(* IEC 61131-3 sources: RL_MAR/experiments/results/ablation/Ablation_no_post_process_deepseek-ai_DeepSeek-V3.2_20260602_235132, 94 files *)

(* ---- hard_92.st ---- *)
TYPE
    ST_BreakerStatus :
    STRUCT
        Opened : BOOL;
        Closed : BOOL;
    END_STRUCT;

    ST_BreakerControl :
    STRUCT
        Trip : BOOL;
        Close : BOOL;
    END_STRUCT;

    ST_BreakerData :
    STRUCT
        Control : ST_BreakerControl;
        Status : ST_BreakerStatus;
    END_STRUCT;

    ST_PointData :
    STRUCT
        Point_1a : INT;
        Point_2a : INT;
        Point_3a : INT;
        Point_4a : INT;
    END_STRUCT;

    E_BreakerID :
    (
        B10_1,
        B10_2,
        B10_12,
        B54,
        B55,
        B56,
        B57
    );
END_TYPE

FUNCTION_BLOCK FB_BreakerControlSystem
VAR_INPUT
    B10_1_Trip : BOOL;
    B10_1_Close : BOOL;
    B10_2_Trip : BOOL;
    B10_2_Close : BOOL;
    B10_12_Trip : BOOL;
    B10_12_Close : BOOL;
    B54_Trip : BOOL;
    B54_Close : BOOL;
    B55_Trip : BOOL;
    B55_Close : BOOL;
    B56_Trip : BOOL;
    B56_Close : BOOL;
    B57_Trip : BOOL;
    B57_Close : BOOL;
END_VAR

VAR_OUTPUT
    Point_1a : INT;
    Point_2a : INT;
    Point_3a : INT;
    Point_4a : INT;
    B10_1_Opened : BOOL;
    B10_1_Closed : BOOL;
    B10_2_Opened : BOOL;
    B10_2_Closed : BOOL;
    B10_12_Opened : BOOL;
    B10_12_Closed : BOOL;
    B54_Opened : BOOL;
    B54_Closed : BOOL;
    B55_Opened : BOOL;
    B55_Closed : BOOL;
    B56_Opened : BOOL;
    B56_Closed : BOOL;
    B57_Opened : BOOL;
    B57_Closed : BOOL;
END_VAR

VAR
    // Internal structured data storage for breakers and points
    rBreakers : ARRAY[E_BreakerID] OF ST_BreakerData;
    rPoints : ST_PointData;
    // Intermediate condition variables
    bCondition_1A : BOOL;
    bCondition_2A : BOOL;
    // Internal variables as per original specification (initialized but not used in core logic)
    SEL86_OUT : INT;
    MOVE89_OUT : INT;
    SEL66_OUT : INT;
    MOVE69_OUT : INT;
    SEL96_OUT : INT;
    MOVE99_OUT : INT;
    SEL106_OUT : INT;
    MOVE109_OUT : INT;
END_VAR

// Main Execution Logic
// Step 1: Update all breaker states based on control signals
// Breaker B10_1
IF rBreakers[B10_1].Control.Close <> B10_1_Close THEN
    rBreakers[B10_1].Control.Close := B10_1_Close;
END_IF;
IF rBreakers[B10_1].Control.Trip <> B10_1_Trip THEN
    rBreakers[B10_1].Control.Trip := B10_1_Trip;
END_IF;

IF B10_1_Close THEN
    rBreakers[B10_1].Status.Closed := TRUE;
    rBreakers[B10_1].Status.Opened := FALSE;
ELSIF B10_1_Trip THEN
    rBreakers[B10_1].Status.Closed := FALSE;
    rBreakers[B10_1].Status.Opened := TRUE;
END_IF;

// Breaker B10_2
IF rBreakers[B10_2].Control.Close <> B10_2_Close THEN
    rBreakers[B10_2].Control.Close := B10_2_Close;
END_IF;
IF rBreakers[B10_2].Control.Trip <> B10_2_Trip THEN
    rBreakers[B10_2].Control.Trip := B10_2_Trip;
END_IF;

IF B10_2_Close THEN
    rBreakers[B10_2].Status.Closed := TRUE;
    rBreakers[B10_2].Status.Opened := FALSE;
ELSIF B10_2_Trip THEN
    rBreakers[B10_2].Status.Closed := FALSE;
    rBreakers[B10_2].Status.Opened := TRUE;
END_IF;

// Breaker B10_12
IF rBreakers[B10_12].Control.Close <> B10_12_Close THEN
    rBreakers[B10_12].Control.Close := B10_12_Close;
END_IF;
IF rBreakers[B10_12].Control.Trip <> B10_12_Trip THEN
    rBreakers[B10_12].Control.Trip := B10_12_Trip;
END_IF;

IF B10_12_Close THEN
    rBreakers[B10_12].Status.Closed := TRUE;
    rBreakers[B10_12].Status.Opened := FALSE;
ELSIF B10_12_Trip THEN
    rBreakers[B10_12].Status.Closed := FALSE;
    rBreakers[B10_12].Status.Opened := TRUE;
END_IF;

// Breaker B54
IF rBreakers[B54].Control.Close <> B54_Close THEN
    rBreakers[B54].Control.Close := B54_Close;
END_IF;
IF rBreakers[B54].Control.Trip <> B54_Trip THEN
    rBreakers[B54].Control.Trip := B54_Trip;
END_IF;

IF B54_Close THEN
    rBreakers[B54].Status.Closed := TRUE;
    rBreakers[B54].Status.Opened := FALSE;
ELSIF B54_Trip THEN
    rBreakers[B54].Status.Closed := FALSE;
    rBreakers[B54].Status.Opened := TRUE;
END_IF;

// Breaker B55
IF rBreakers[B55].Control.Close <> B55_Close THEN
    rBreakers[B55].Control.Close := B55_Close;
END_IF;
IF rBreakers[B55].Control.Trip <> B55_Trip THEN
    rBreakers[B55].Control.Trip := B55_Trip;
END_IF;

IF B55_Close THEN
    rBreakers[B55].Status.Closed := TRUE;
    rBreakers[B55].Status.Opened := FALSE;
ELSIF B55_Trip THEN
    rBreakers[B55].Status.Closed := FALSE;
    rBreakers[B55].Status.Opened := TRUE;
END_IF;

// Breaker B56
IF rBreakers[B56].Control.Close <> B56_Close THEN
    rBreakers[B56].Control.Close := B56_Close;
END_IF;
IF rBreakers[B56].Control.Trip <> B56_Trip THEN
    rBreakers[B56].Control.Trip := B56_Trip;
END_IF;

IF B56_Close THEN
    rBreakers[B56].Status.Closed := TRUE;
    rBreakers[B56].Status.Opened := FALSE;
ELSIF B56_Trip THEN
    rBreakers[B56].Status.Closed := FALSE;
    rBreakers[B56].Status.Opened := TRUE;
END_IF;

// Breaker B57
IF rBreakers[B57].Control.Close <> B57_Close THEN
    rBreakers[B57].Control.Close := B57_Close;
END_IF;
IF rBreakers[B57].Control.Trip <> B57_Trip THEN
    rBreakers[B57].Control.Trip := B57_Trip;
END_IF;

IF B57_Close THEN
    rBreakers[B57].Status.Closed := TRUE;
    rBreakers[B57].Status.Opened := FALSE;
ELSIF B57_Trip THEN
    rBreakers[B57].Status.Closed := FALSE;
    rBreakers[B57].Status.Opened := TRUE;
END_IF;

// Step 2: Calculate intermediate conditions
bCondition_1A := (rBreakers[B10_12].Status.Closed AND rBreakers[B10_1].Status.Closed) OR rBreakers[B10_2].Status.Closed;
bCondition_2A := (rBreakers[B10_12].Status.Closed AND rBreakers[B10_2].Status.Closed) OR rBreakers[B10_1].Status.Closed;

// Step 3: Calculate output points
// Point_1a
IF rBreakers[B54].Status.Closed AND bCondition_1A THEN
    rPoints.Point_1a := 0;
ELSE
    rPoints.Point_1a := 138;
END_IF;

// Point_2a
IF rBreakers[B55].Status.Closed AND bCondition_1A THEN
    rPoints.Point_2a := 0;
ELSE
    rPoints.Point_2a := 138;
END_IF;

// Point_3a
IF rBreakers[B56].Status.Closed AND bCondition_2A THEN
    rPoints.Point_3a := 0;
ELSE
    rPoints.Point_3a := 138;
END_IF;

// Point_4a
IF rBreakers[B57].Status.Closed AND bCondition_2A THEN
    rPoints.Point_4a := 0;
ELSE
    rPoints.Point_4a := 138;
END_IF;

// Step 4: Map internal data to public outputs
Point_1a := rPoints.Point_1a;
Point_2a := rPoints.Point_2a;
Point_3a := rPoints.Point_3a;
Point_4a := rPoints.Point_4a;

B10_1_Opened := rBreakers[B10_1].Status.Opened;
B10_1_Closed := rBreakers[B10_1].Status.Closed;
B10_2_Opened := rBreakers[B10_2].Status.Opened;
B10_2_Closed := rBreakers[B10_2].Status.Closed;
B10_12_Opened := rBreakers[B10_12].Status.Opened;
B10_12_Closed := rBreakers[B10_12].Status.Closed;
B54_Opened := rBreakers[B54].Status.Opened;
B54_Closed := rBreakers[B54].Status.Closed;
B55_Opened := rBreakers[B55].Status.Opened;
B55_Closed := rBreakers[B55].Status.Closed;
B56_Opened := rBreakers[B56].Status.Opened;
B56_Closed := rBreakers[B56].Status.Closed;
B57_Opened := rBreakers[B57].Status.Opened;
B57_Closed := rBreakers[B57].Status.Closed;

// Step 5: Initialize internal placeholder variables (as per original spec)
SEL86_OUT := 0;
MOVE89_OUT := 0;
SEL66_OUT := 0;
MOVE69_OUT := 0;
SEL96_OUT := 0;
MOVE99_OUT := 0;
SEL106_OUT := 0;
MOVE109_OUT := 0;

END_FUNCTION_BLOCK

(* ---- hard_93.st ---- *)
FUNCTION_BLOCK FB_CircuitControl
VAR_INPUT
    Reset_All_CB : BOOL;
    Current_Fault_on_TRSF1 : INT;
    Current_Fault_on_66BUS1 : INT;
END_VAR

VAR_OUTPUT
    Short_Circuit_TRSF1 : BOOL;
    Short_Circuit_66BUS : BOOL;
    Open_CB1_66KV : BOOL;
    Open_CB2_66KV : BOOL;
    Open_CB_TRSF1 : BOOL;
    Open_CB2_22KV : BOOL;
END_VAR

VAR
    Threshold500 : INT := 500;
    Prev_Open_CB2_22KV : BOOL;
    Prev_Open_CB1_66KV : BOOL;
    Prev_Open_CB_TRSF1 : BOOL;
    bTemp_Open_CB2_22KV : BOOL;
    bTemp_Open_CB1_66KV : BOOL;
    bTemp_Open_CB_TRSF1 : BOOL;
END_VAR

(* Part a: Short circuit detection *)
Short_Circuit_66BUS := (Current_Fault_on_66BUS1 > Threshold500);
Short_Circuit_TRSF1 := (Current_Fault_on_TRSF1 > Threshold500);

(* Part b: Circuit breaker control logic *)
(* Reset condition takes highest priority *)
IF Reset_All_CB THEN
    Open_CB1_66KV := FALSE;
    Open_CB2_66KV := FALSE;
    Open_CB_TRSF1 := FALSE;
    Open_CB2_22KV := FALSE;
    Prev_Open_CB2_22KV := FALSE;
    Prev_Open_CB1_66KV := FALSE;
    Prev_Open_CB_TRSF1 := FALSE;
ELSE
    (* Open_CB2_66KV is always TRUE (closed) per specification *)
    Open_CB2_66KV := TRUE;

    (* First pass: Initial calculations using previous cycle states *)
    bTemp_Open_CB2_22KV := (NOT Prev_Open_CB2_22KV) AND
                           ((Open_CB1_66KV AND Open_CB_TRSF1) OR Short_Circuit_66BUS);

    bTemp_Open_CB1_66KV := (NOT bTemp_Open_CB2_22KV) AND
                           ((Prev_Open_CB1_66KV AND Open_CB_TRSF1) OR Short_Circuit_66BUS);

    bTemp_Open_CB_TRSF1 := (NOT bTemp_Open_CB2_22KV) AND
                           ((Open_CB1_66KV AND Prev_Open_CB_TRSF1) OR Short_Circuit_66BUS);

    (* Second pass: Update calculations using intermediate values *)
    bTemp_Open_CB2_22KV := bTemp_Open_CB2_22KV OR
                          ((NOT Prev_Open_CB2_22KV) AND
                           ((Open_CB2_66KV AND bTemp_Open_CB1_66KV AND bTemp_Open_CB_TRSF1) OR Short_Circuit_TRSF1));

    bTemp_Open_CB1_66KV := bTemp_Open_CB1_66KV OR
                          ((NOT bTemp_Open_CB2_22KV) AND
                           ((Open_CB2_66KV AND Prev_Open_CB1_66KV AND bTemp_Open_CB_TRSF1) OR Short_Circuit_TRSF1));

    bTemp_Open_CB_TRSF1 := bTemp_Open_CB_TRSF1 OR
                          ((NOT bTemp_Open_CB2_22KV) AND
                           ((Open_CB2_66KV AND bTemp_Open_CB1_66KV AND Prev_Open_CB_TRSF1) OR Short_Circuit_TRSF1));

    (* Assign final values to outputs *)
    Open_CB2_22KV := bTemp_Open_CB2_22KV;
    Open_CB1_66KV := bTemp_Open_CB1_66KV;
    Open_CB_TRSF1 := bTemp_Open_CB_TRSF1;

    (* Store current states for next scan cycle *)
    Prev_Open_CB2_22KV := Open_CB2_22KV;
    Prev_Open_CB1_66KV := Open_CB1_66KV;
    Prev_Open_CB_TRSF1 := Open_CB_TRSF1;
END_IF;

END_FUNCTION_BLOCK;

(* ---- hard_94.st ---- *)
FUNCTION_BLOCK FB_AdvancedCircuitBreakerControl
VAR_INPUT
    S_AL1_P_B1 : BOOL;
    S_AL1_P_B2 : BOOL;
    S_AL1_MCB : BOOL;
    MCB_BUSY : BOOL;
    MCB_ERROR : BOOL;
    S_AL1_MCBR : BOOL;
    MCBR_BUSY : BOOL;
    MCBR_ERROR : BOOL;
    S_AL1_P_B3 : BOOL;
    S_AL1_MCB2 : BOOL;
    S_AL1_MCBR2 : BOOL;
END_VAR
VAR_OUTPUT
    E_AL1_B1 : BOOL;
    PUWS_AL1_B1_PLUS : BOOL;
    PUWS_AL1_B1_RIGHT : BOOL;
    PAS_AL1_PLUS : BOOL;
    PAS_AL1_TURN : BOOL;
END_VAR
VAR
    (* State Variables - Only one should be active at a time *)
    PPAL1 : BOOL := 1;
    PP0 : BOOL := 0;
    PP1 : BOOL := 0;
    PP2 : BOOL := 0;
    PP3 : BOOL := 0;
    PP4 : BOOL := 0;
    PP5 : BOOL := 0;
    PP7 : BOOL := 0;
    PPL3 : BOOL := 0;
    PPL4 : BOOL := 0;
    PPL5 : BOOL := 0;
    PPL7 : BOOL := 0;

    (* Internal Control and Status Flags *)
    MCB : BOOL := 1;
    MCBR : BOOL := 1;
    MCB_CONTROL : BOOL;
    STABLE : BOOL;
END_VAR

(* Main State Machine Logic *)
STABLE := 0;
WHILE (STABLE = 0) DO
    STABLE := 1;

    (* State PP0 to PP1 *)
    IF (PP0 = 1) AND (NOT MCB_CONTROL) AND (PP1 = 0) THEN
        PP0 := 0;
        PP1 := 1;
        STABLE := 0;
    END_IF;

    (* State PP1 to PP2 *)
    IF (PP1 = 1) AND S_AL1_P_B1 AND (PP2 = 0) THEN
        PP1 := 0;
        PP2 := 1;
        STABLE := 0;
    END_IF;

    (* State PP2 to PP3 (Main Path) *)
    IF (PP2 = 1) AND S_AL1_P_B2 AND (NOT MCB_CONTROL) AND (PP3 = 0) THEN
        PP2 := 0;
        PP3 := 1;
        STABLE := 0;
    END_IF;

    (* State PP2 to PPL3 (Alternative Path) *)
    IF (PP2 = 1) AND S_AL1_P_B2 AND MCB_CONTROL AND (PPL3 = 0) AND (PP1 = 0) THEN
        PP2 := 0;
        PPL3 := 1;
        PP1 := 1;
        STABLE := 0;
    END_IF;

    (* State PP3 to PP4 *)
    IF (PP3 = 1) AND S_AL1_MCB AND (PP4 = 0) AND (PP1 = 0) THEN
        PP3 := 0;
        PP4 := 1;
        PP1 := 1;
        STABLE := 0;
    END_IF;

    (* State PP4 to PP5 *)
    IF (PP4 = 1) AND (MCB = 1) AND MCB_BUSY AND (PP5 = 0) THEN
        PP4 := 0;
        MCB := 0;
        PP5 := 1;
        STABLE := 0;
    END_IF;

    (* State PP5 to PP7 *)
    IF (PP5 = 1) AND S_AL1_MCB2 AND (PP7 = 0) AND (MCB = 0) THEN
        PP5 := 0;
        PP7 := 1;
        MCB := 1;
        STABLE := 0;
    END_IF;

    (* State PP7 to End *)
    IF (PP7 = 1) AND S_AL1_P_B3 THEN
        PP7 := 0;
        STABLE := 0;
    END_IF;

    (* State PPL3 to PPL4 *)
    IF (PPL3 = 1) AND S_AL1_MCBR AND (PPL4 = 0) THEN
        PPL3 := 0;
        PPL4 := 1;
        STABLE := 0;
    END_IF;

    (* State PPL4 to PPL5 *)
    IF (PPL4 = 1) AND (MCBR = 1) AND MCBR_BUSY AND (PPL5 = 0) THEN
        PPL4 := 0;
        MCBR := 0;
        PPL5 := 1;
        STABLE := 0;
    END_IF;

    (* State PPL5 to PPL7 *)
    IF (PPL5 = 1) AND S_AL1_MCBR2 AND (PPL7 = 0) AND (MCBR = 0) THEN
        PPL5 := 0;
        PPL7 := 1;
        MCBR := 1;
        STABLE := 0;
    END_IF;

    (* State PPL7 to End *)
    IF (PPL7 = 1) AND S_AL1_P_B3 THEN
        PPL7 := 0;
        STABLE := 0;
    END_IF;
END_WHILE;

(* Output Control Logic *)
(* Initialize all outputs to FALSE *)
E_AL1_B1 := 0;
PUWS_AL1_B1_PLUS := 0;
PUWS_AL1_B1_RIGHT := 0;
PAS_AL1_PLUS := 0;
PAS_AL1_TURN := 0;
MCB_CONTROL := 0;

(* Set outputs based on active states *)
IF (PP0 = 1) OR (PP1 = 1) THEN
    E_AL1_B1 := 1;
END_IF;

IF (PP3 = 1) THEN
    MCB_CONTROL := 1;
END_IF;

IF (PPL3 = 1) OR (PPL4 = 1) THEN
    PAS_AL1_PLUS := 1;
    PAS_AL1_TURN := 1;
END_IF;

IF (PPAL1 = 1) OR (PP2 = 1) THEN
    PUWS_AL1_B1_PLUS := 1;
END_IF;

IF (PP2 = 1) OR (PP3 = 1) OR (PPL3 = 1) THEN
    E_AL1_B1 := 0;
END_IF;

IF (PP0 = 1) OR (PP3 = 1) THEN
    MCB_CONTROL := 0;
END_IF;

IF (PP0 = 1) OR (PP3 = 1) OR (PP4 = 1) THEN
    PAS_AL1_PLUS := 0;
    PAS_AL1_TURN := 0;
END_IF;

IF (PPAL1 = 1) OR (PP2 = 1) THEN
    PUWS_AL1_B1_RIGHT := 0;
END_IF;

END_FUNCTION_BLOCK

(* ---- hf_1.st ---- *)
FUNCTION_BLOCK StackMin
VAR_INPUT
    push : BOOL;
    pop : BOOL;
    reset : BOOL;
END_VAR
VAR_OUTPUT
    error : BOOL;
    status : WORD;
END_VAR
VAR_IN_OUT
    item : INT;
    stack : ARRAY[0..3] OF INT;
END_VAR
VAR
    top : INT := -1;
    i : INT;
    minIndex : INT;
    minValue : INT;
END_VAR

(* Reset has highest priority *)
IF reset THEN
    top := -1;
    error := FALSE;
    status := 16#0000;
ELSIF push THEN
    (* Push operation *)
    IF top >= 3 THEN
        error := TRUE;
        status := 16#8A04;
    ELSE
        top := top + 1;
        stack[top] := item;
        error := FALSE;
        status := 16#0000;
    END_IF;
ELSIF pop THEN
    (* Pop-minimum operation *)
    IF top < 0 THEN
        error := TRUE;
        status := 16#8A05;
    ELSE
        (* Find minimum value and its index *)
        minIndex := 0;
        minValue := stack[0];
        FOR i := 1 TO top DO
            IF stack[i] < minValue THEN
                minValue := stack[i];
                minIndex := i;
            END_IF;
        END_FOR;

        (* Output the minimum value *)
        item := minValue;

        (* Shift elements down to remove the minimum *)
        FOR i := minIndex TO top - 1 DO
            stack[i] := stack[i + 1];
        END_FOR;

        (* Decrement top index *)
        top := top - 1;

        error := FALSE;
        status := 16#0000;
    END_IF;
ELSE
    (* No operation - maintain current state *)
    error := FALSE;
    status := 16#0000;
END_IF;

END_FUNCTION_BLOCK

(* ---- hf_10.st ---- *)
TYPE
    // Define a circular buffer structure for clarity and maintainability
    CircularBuffer : STRUCT
        Data : ARRAY[1..100] OF REAL;
        Head : INT; // Points to the oldest element (next to be overwritten)
        Count : INT; // Number of valid elements currently in the buffer
        Sum : REAL;
    END_STRUCT;
END_TYPE

FUNCTION_BLOCK FloatingAverage
VAR_INPUT
    cyclicExecution : BOOL; // When TRUE, periodic reading is performed, and trigger has no effect
    trigger : BOOL; // External trigger signal, reads value upon each rising edge
    value : REAL; // Newly read data value
    windowSize : INT; // The window size for the moving average, which must be between 1 and 100
    reset : BOOL; // Reset signal, resets the moving average calculation when TRUE
END_VAR
VAR_OUTPUT
    average : REAL; // The moving average
    windowSizeReached : BOOL; // FALSE: Maximum window width not yet reached, TRUE: Maximum window width has been reached
    error : BOOL; // FALSE: No error occurred, TRUE: An error occurred during the execution of FB
    status : WORD; // Status code
END_VAR
VAR
    // Internal state variables
    Buffer : CircularBuffer;
    triggerPrev : BOOL := FALSE;
    windowSizeInternal : INT := 1;
    // Constants for status codes
    STATUS_OK : WORD := 16#0000;
    STATUS_WINDOW_ERROR : WORD := 16#8200;
END_VAR

// ========== MAIN LOGIC ==========

// 1. Handle RESET signal with highest priority
IF reset THEN
    // Reset the internal buffer state
    Buffer.Head := 1;
    Buffer.Count := 0;
    Buffer.Sum := 0.0;
    // Clear the buffer array (optional for clarity, but Count=0 makes them irrelevant)
    FOR i := 1 TO 100 DO
        Buffer.Data[i] := 0.0;
    END_FOR;

    // Reset outputs
    average := 0.0;
    windowSizeReached := FALSE;
    error := FALSE;
    status := STATUS_OK;

    // Reset internal tracking
    windowSizeInternal := 1;
    triggerPrev := FALSE;

    RETURN; // Exit the function block, no further processing this cycle
END_IF;

// 2. Validate windowSize on EVERY execution (not just on reset)
IF (windowSize < 1) OR (windowSize > 100) THEN
    // Set error state, do NOT process any new data
    error := TRUE;
    status := STATUS_WINDOW_ERROR;
    average := 0.0;
    windowSizeReached := FALSE;

    // Preserve internal state (no updates)
    triggerPrev := trigger; // Still update edge detection to avoid stuck trigger
    RETURN; // Exit the function block, no further processing this cycle
ELSE
    // Window size is valid, clear any previous error
    error := FALSE;
    status := STATUS_OK;
    windowSizeInternal := windowSize; // Store the valid size for internal use
END_IF;

// 3. Determine if a new value should be processed
//    Priority: cyclicExecution overrides trigger
IF cyclicExecution THEN
    // Process the new value immediately in cyclic mode
    ProcessNewValue(value);
ELSIF trigger AND NOT triggerPrev THEN
    // Process the new value on the rising edge of trigger
    ProcessNewValue(value);
END_IF;

// 4. Update edge detection for the trigger signal
triggerPrev := trigger;

// 5. Calculate and set the output average
IF Buffer.Count > 0 THEN
    average := Buffer.Sum / INT_TO_REAL(Buffer.Count);
ELSE
    average := 0.0;
END_IF;

// 6. Set the windowSizeReached flag
windowSizeReached := (Buffer.Count >= windowSizeInternal);

// ========== INTERNAL FUNCTION ==========
// Encapsulates the core buffer update logic for clarity and reuse
METHOD ProcessNewValue : BOOL
VAR_INPUT
    newValue : REAL;
END_VAR
VAR
    oldestValue : REAL;
END_VAR

    // If buffer is already at full window size, we need to remove the oldest value
    IF Buffer.Count >= windowSizeInternal THEN
        // The oldest value is at the current Head position
        oldestValue := Buffer.Data[Buffer.Head];
        Buffer.Sum := Buffer.Sum - oldestValue;

        // Overwrite the oldest value with the new one
        Buffer.Data[Buffer.Head] := newValue;
        Buffer.Sum := Buffer.Sum + newValue;

        // Move Head to the next position (circular)
        Buffer.Head := Buffer.Head + 1;
        IF Buffer.Head > windowSizeInternal THEN
            Buffer.Head := 1;
        END_IF;
        // Count remains unchanged (windowSizeInternal)
    ELSE
        // Buffer is not yet full, simply add the new value
        // Insert at position: Head + Count (since Head points to first element when full)
        // When not full, we can just append sequentially
        Buffer.Count := Buffer.Count + 1;
        Buffer.Data[Buffer.Count] := newValue;
        Buffer.Sum := Buffer.Sum + newValue;
        // Head remains at 1 until the buffer fills for the first time
    END_IF;

    ProcessNewValue := TRUE; // Success
END_METHOD

END_FUNCTION_BLOCK;

(* ---- hf_11.st ---- *)
FUNCTION_BLOCK FB_BottleProcessing
VAR_INPUT
    bottleSensor : BOOL;
    cleaningConfirmButton : BOOL;
    fillingConfirmButton : BOOL;
    cappingConfirmButton : BOOL;
    packingConfirmButton : BOOL;
    finishedButton : BOOL;
END_VAR

VAR_OUTPUT
    Pump_Motor : BOOL;
    Filling_Valve : BOOL;
    Capping_Machine : BOOL;
    Packing_Machine : BOOL;
    Completion_Light : BOOL;
END_VAR

VAR
    State : INT := 0; (* 0=Waiting, 1=Cleaning, 2=Filling, 3=Capping, 4=Packing, 5=Completed *)
END_VAR

CASE State OF
    0: (* Waiting *)
        IF bottleSensor THEN
            Pump_Motor := TRUE;
            State := 1;
        END_IF;

    1: (* Cleaning *)
        IF cleaningConfirmButton THEN
            Pump_Motor := FALSE;
            Filling_Valve := TRUE;
            State := 2;
        END_IF;

    2: (* Filling *)
        IF fillingConfirmButton THEN
            Filling_Valve := FALSE;
            Capping_Machine := TRUE;
            State := 3;
        END_IF;

    3: (* Capping *)
        IF cappingConfirmButton THEN
            Capping_Machine := FALSE;
            Packing_Machine := TRUE;
            State := 4;
        END_IF;

    4: (* Packing *)
        IF packingConfirmButton THEN
            Packing_Machine := FALSE;
            Completion_Light := TRUE;
            State := 5;
        END_IF;

    5: (* Completed *)
        IF finishedButton THEN
            Completion_Light := FALSE;
            Pump_Motor := FALSE;
            Filling_Valve := FALSE;
            Capping_Machine := FALSE;
            Packing_Machine := FALSE;
            State := 0;
        END_IF;
END_CASE;
END_FUNCTION_BLOCK

(* ---- hf_12.st ---- *)
FUNCTION_BLOCK MaterialMixing
VAR_INPUT
    estop : BOOL; (* Emergency Stop Signal, FALSE: Emergency stop triggered, TRUE: No emergency stop triggered *)
    opeMode : BOOL; (* Operation Mode, FALSE: Manual Operation Mode, TRUE: Automatic Operation Mode *)
    valveAStart : BOOL; (* Valve A Start Button *)
    valveBStart : BOOL; (* Valve B Start Button *)
    valveCStart : BOOL; (* Valve C Start Button *)
    valveDStart : BOOL; (* Valve D Start Button *)
    mixMotorStart : BOOL; (* Mixing Motor Start Button *)
    autoStart : BOOL; (* Automatic Start Button *)
    processMode : BOOL; (* Process Mode *)
    levelSensor : INT; (* Liquid Level Sensor, unit cm *)
    mixMotorComplete : BOOL; (* Mixing Complete Signal *)
END_VAR

VAR_OUTPUT
    valveARun : BOOL; (* Valve A Run Command *)
    valveBRun : BOOL; (* Valve B Run Command *)
    valveCRun : BOOL; (* Valve C Run Command *)
    valveDRun : BOOL; (* Valve D Run Command *)
    mixMotorRun : BOOL; (* Mixing Motor Run Command *)
END_VAR

VAR
    (* Edge detection for manual mode buttons *)
    previousValveAStart : BOOL := FALSE;
    previousValveBStart : BOOL := FALSE;
    previousValveCStart : BOOL := FALSE;
    previousValveDStart : BOOL := FALSE;
    previousMixMotorStart : BOOL := FALSE;
    previousAutoStart : BOOL := FALSE;

    (* Automatic process state variables *)
    autoProcessActive : BOOL := FALSE;
    autoStep : INT := 0;

    (* Safety level interlock constant *)
    MAX_SAFE_LEVEL : INT := 105;
END_VAR

(* --- Primary Safety Logic: Emergency Stop & Overfill Protection --- *)
IF NOT estop THEN
    (* Emergency Stop Active: De-energize all outputs and reset automatic process *)
    valveARun := FALSE;
    valveBRun := FALSE;
    valveCRun := FALSE;
    valveDRun := FALSE;
    mixMotorRun := FALSE;
    autoProcessActive := FALSE;
    autoStep := 0;
ELSE
    (* Emergency Stop NOT Active: Normal Operation *)

    (* Independent Safety Interlock: Prevent overfilling *)
    IF levelSensor >= MAX_SAFE_LEVEL THEN
        valveARun := FALSE;
        valveBRun := FALSE;
        valveCRun := FALSE;
    END_IF;

    (* --- Mode Selection --- *)
    IF opeMode THEN
        (* --- AUTOMATIC MODE --- *)

        (* Toggle automatic process on rising edge of autoStart *)
        IF autoStart AND NOT previousAutoStart THEN
            autoProcessActive := NOT autoProcessActive;
            IF autoProcessActive THEN
                autoStep := 1; (* Start sequence *)
            ELSE
                autoStep := 0; (* Abort sequence *)
            END_IF;
        END_IF;
        previousAutoStart := autoStart;

        (* Automatic Process Sequence *)
        IF autoProcessActive THEN
            CASE autoStep OF
                1: (* Step 1: Open Valve A *)
                    valveARun := TRUE;
                    IF levelSensor >= 50 THEN
                        valveARun := FALSE;
                        autoStep := 2;
                    END_IF;

                2: (* Step 2: Open Valve B *)
                    valveBRun := TRUE;
                    IF levelSensor >= 80 THEN
                        valveBRun := FALSE;
                        autoStep := 3;
                    END_IF;

                3: (* Step 3: Branch based on processMode *)
                    IF NOT processMode THEN
                        (* Path for processMode = FALSE: Start Mixing *)
                        mixMotorRun := TRUE;
                        IF mixMotorComplete THEN
                            mixMotorRun := FALSE;
                            autoStep := 5; (* Skip to Valve D *)
                        END_IF;
                    ELSE
                        (* Path for processMode = TRUE: Open Valve C *)
                        valveCRun := TRUE;
                        IF levelSensor >= 100 THEN
                            valveCRun := FALSE;
                            autoStep := 4;
                        END_IF;
                    END_IF;

                4: (* Step 4: Mixing for processMode = TRUE path *)
                    mixMotorRun := TRUE;
                    IF mixMotorComplete THEN
                        mixMotorRun := FALSE;
                        autoStep := 5;
                    END_IF;

                5: (* Step 5: Open Valve D and end sequence *)
                    valveDRun := TRUE;
                    autoProcessActive := FALSE;
                    autoStep := 0;
            END_CASE;
        ELSE
            (* Automatic process not active: ensure all outputs are off *)
            valveARun := FALSE;
            valveBRun := FALSE;
            valveCRun := FALSE;
            valveDRun := FALSE;
            mixMotorRun := FALSE;
        END_IF;

    ELSE
        (* --- MANUAL MODE --- *)

        (* Valve A: Toggle on rising edge *)
        IF valveAStart AND NOT previousValveAStart THEN
            valveARun := NOT valveARun;
        END_IF;
        previousValveAStart := valveAStart;

        (* Valve B: Toggle on rising edge *)
        IF valveBStart AND NOT previousValveBStart THEN
            valveBRun := NOT valveBRun;
        END_IF;
        previousValveBStart := valveBStart;

        (* Valve C: Toggle on rising edge *)
        IF valveCStart AND NOT previousValveCStart THEN
            valveCRun := NOT valveCRun;
        END_IF;
        previousValveCStart := valveCStart;

        (* Valve D: Toggle on rising edge *)
        IF valveDStart AND NOT previousValveDStart THEN
            valveDRun := NOT valveDRun;
        END_IF;
        previousValveDStart := valveDStart;

        (* Mixing Motor: Toggle on rising edge *)
        IF mixMotorStart AND NOT previousMixMotorStart THEN
            mixMotorRun := NOT mixMotorRun;
        END_IF;
        previousMixMotorStart := mixMotorStart;
    END_IF;
END_IF;

END_FUNCTION_BLOCK;

(* ---- hf_13.st ---- *)
(* Custom TON Timer Function Block for Single-Cycle Execution Model *)
FUNCTION_BLOCK TON
VAR_INPUT
    IN : BOOL;
    PT : DINT;
    CYCLE_TIME : DINT;
END_VAR
VAR_OUTPUT
    Q : BOOL;
    ET : DINT;
END_VAR
VAR
    elapsedTimeInternal : DINT := 0;
    IN_PREV : BOOL := FALSE;
END_VAR

IF IN THEN
    IF NOT IN_PREV THEN
        elapsedTimeInternal := 0;
    END_IF;

    IF elapsedTimeInternal < PT THEN
        elapsedTimeInternal := elapsedTimeInternal + CYCLE_TIME;
        Q := FALSE;
    ELSE
        elapsedTimeInternal := PT;
        Q := TRUE;
    END_IF;

    ET := elapsedTimeInternal;
ELSE
    Q := FALSE;
    ET := 0;
    elapsedTimeInternal := 0;
END_IF;

IN_PREV := IN;
END_FUNCTION_BLOCK

(* Main Lights Control Function Block *)
FUNCTION_BLOCK LightsControl
VAR_INPUT
    button1 : BOOL; (* Button 1: Automatic/Manual Mode Select *)
    button2 : BOOL; (* Button 2: Manual Control/Green Light Req *)
    button3 : BOOL; (* Button 3: Manual Control/Red Light Req *)
    CYCLE_TIME : DINT; (* Time elapsed in current cycle (in ms) *)
END_VAR
VAR_OUTPUT
    greenLight : BOOL; (* Green light *)
    redLight : BOOL; (* Red light *)
    yellowLight : BOOL; (* Yellow light *)
END_VAR
VAR
    (* Timers for control *)
    timerAuto : TON;
    timerGreen : TON;
    timerRed : TON;
    timerYellow : TON;

    currentState : INT := 0;
    autoRunTimer : BOOL;
END_VAR

(* Reset manual timers at start of every PLC cycle as required *)
timerGreen.IN := FALSE;
timerGreen.PT := 1000;
timerGreen.CYCLE_TIME := CYCLE_TIME;

timerRed.IN := FALSE;
timerRed.PT := 2000;
timerRed.CYCLE_TIME := CYCLE_TIME;

timerYellow.IN := FALSE;
timerYellow.PT := 1000;
timerYellow.CYCLE_TIME := CYCLE_TIME;

(* Main mode selection *)
IF button1 THEN
    (* Automatic Mode *)
    timerAuto.IN := TRUE;
    timerAuto.PT := 1000;
    timerAuto.CYCLE_TIME := CYCLE_TIME;
    timerAuto();

    (* State machine logic *)
    IF timerAuto.Q THEN
        currentState := currentState + 1;
        IF currentState >= 3 THEN
            currentState := 0;
        END_IF;
    END_IF;

    (* Set outputs based on current state *)
    CASE currentState OF
        0: (* State 0: Green light on for 1 second *)
            greenLight := TRUE;
            redLight := FALSE;
            yellowLight := FALSE;

        1: (* State 1: Red light on for 1 second *)
            greenLight := FALSE;
            redLight := TRUE;
            yellowLight := FALSE;

        2: (* State 2: Yellow light on for 1 second *)
            greenLight := FALSE;
            redLight := FALSE;
            yellowLight := TRUE;
    END_CASE;
ELSE
    (* Manual Mode *)
    timerAuto.IN := FALSE;

    (* Evaluate button combinations *)
    IF NOT button2 AND NOT button3 THEN
        (* Both FALSE: All lights off *)
        greenLight := FALSE;
        redLight := FALSE;
        yellowLight := FALSE;

    ELSIF button2 AND NOT button3 THEN
        (* button2 TRUE, button3 FALSE *)
        greenLight := TRUE;
        timerRed.IN := TRUE;
        timerRed();
        redLight := timerRed.Q; (* Blinks at 0.5Hz *)
        yellowLight := FALSE;

    ELSIF NOT button2 AND button3 THEN
        (* button2 FALSE, button3 TRUE *)
        greenLight := FALSE;
        redLight := TRUE;
        timerYellow.IN := TRUE;
        timerYellow();
        yellowLight := NOT timerYellow.Q; (* Blinks at 1Hz *)

    ELSIF button2 AND button3 THEN
        (* Both TRUE *)
        timerGreen.IN := TRUE;
        timerGreen();
        greenLight := NOT timerGreen.Q; (* Blinks at 1Hz *)
        redLight := FALSE;
        yellowLight := TRUE;
    END_IF;
END_IF;
END_FUNCTION_BLOCK

(* ---- hf_14.st ---- *)
TYPE T_GARAGE_SLOT:
STRUCT
    Occupied : BOOL;
    VehicleNumber : INT;
END_STRUCT
END_TYPE

TYPE T_TRUCK_INFO:
STRUCT
    row : INT;
    col : INT;
    VehicleNumber : INT;
END_STRUCT
END_TYPE

FUNCTION_BLOCK TruckGarage
VAR_INPUT
    enter_flag : BOOL;
    exit_flag : BOOL;
    VehicleNumber_in : INT;
END_VAR
VAR_OUTPUT
    truck : T_TRUCK_INFO;
END_VAR
VAR_IN_OUT
    garage : ARRAY[1..3, 1..5] OF T_GARAGE_SLOT;
END_VAR
VAR
    CurrentState : INT; (* 0=IDLE, 1=ENTRY_ALLOCATION, 2=ENTRY_SEARCH, 3=EXIT_SEARCH *)
    i : INT;
    j : INT;
    EntryFound : BOOL;
    ExitFound : BOOL;
END_VAR

(* Main State Machine *)
CASE CurrentState OF
    0: (* IDLE *)
        (* Reset outputs and internal flags *)
        truck.row := 0;
        truck.col := 0;
        truck.VehicleNumber := 0;
        EntryFound := FALSE;
        ExitFound := FALSE;

        (* Determine next state based on request priority *)
        IF enter_flag THEN
            CurrentState := 1; (* Proceed to entry allocation *)
        ELSIF exit_flag THEN
            CurrentState := 3; (* Proceed to exit search *)
        ELSE
            CurrentState := 0; (* Remain idle *)
        END_IF;

    1: (* ENTRY_ALLOCATION - Initialize search for available space *)
        (* Initialize search indices according to "latter row first, latter column first" *)
        i := 3; (* Start from last row *)
        j := 5; (* Start from last column *)
        CurrentState := 2; (* Proceed to search loop *)

    2: (* ENTRY_SEARCH - Find and allocate available parking space *)
        IF (i >= 1) AND (i <= 3) AND (j >= 1) AND (j <= 5) THEN
            IF NOT garage[i, j].Occupied THEN
                (* Found available space - allocate it *)
                garage[i, j].Occupied := TRUE;
                garage[i, j].VehicleNumber := VehicleNumber_in;
                EntryFound := TRUE;
                CurrentState := 0; (* Return to idle *)
            ELSE
                (* Space occupied - move to next position *)
                j := j - 1;
                IF j < 1 THEN
                    (* Move to previous row *)
                    i := i - 1;
                    j := 5;
                    IF i < 1 THEN
                        (* No available spaces found *)
                        CurrentState := 0;
                    END_IF;
                END_IF;
                (* Remain in ENTRY_SEARCH state to continue search *)
            END_IF;
        ELSE
            (* Search indices out of bounds - error recovery *)
            CurrentState := 0;
        END_IF;

    3: (* EXIT_SEARCH - Find and release specified vehicle *)
        (* Initialize search if needed *)
        IF (i < 1) OR (i > 3) OR (j < 1) OR (j > 5) THEN
            i := 1; (* Start from first row *)
            j := 1; (* Start from first column *)
        END_IF;

        IF (i >= 1) AND (i <= 3) AND (j >= 1) AND (j <= 5) THEN
            IF garage[i, j].Occupied AND (garage[i, j].VehicleNumber = VehicleNumber_in) THEN
                (* Found vehicle to exit - release space *)
                truck.row := i;
                truck.col := j;
                truck.VehicleNumber := VehicleNumber_in;
                garage[i, j].Occupied := FALSE;
                garage[i, j].VehicleNumber := 0;
                ExitFound := TRUE;
                CurrentState := 0; (* Return to idle *)
            ELSE
                (* Not the target vehicle - move to next position *)
                (* Follow "former row first, former column first" for search order *)
                j := j + 1;
                IF j > 5 THEN
                    i := i + 1;
                    j := 1;
                    IF i > 3 THEN
                        (* Vehicle not found in garage *)
                        CurrentState := 0;
                    END_IF;
                END_IF;
                (* Remain in EXIT_SEARCH state to continue search *)
            END_IF;
        ELSE
            (* Search indices out of bounds - error recovery *)
            CurrentState := 0;
        END_IF;

    ELSE
        (* Invalid state - reset to IDLE *)
        CurrentState := 0;
END_CASE;

END_FUNCTION_BLOCK

(* ---- hf_15.st ---- *)
FUNCTION_BLOCK FB_MergeBytes
VAR_INPUT
    byteArray : ARRAY[1..20] OF DINT; (* Byte array to be merged *)
END_VAR
VAR_OUTPUT
    dwordArray : ARRAY[1..10] OF DINT; (* Merged double word array *)
    mergeDwordNum : DINT; (* Actual number of merged double words *)
END_VAR
VAR
    i : INT; (* Loop counter for dwordArray clearing *)
    j : INT; (* Loop counter for byte processing within a dword *)
    dwordIdx : INT; (* Current position in dwordArray *)
    byteIdx : INT; (* Current position in byteArray *)
    maxDwordCount : INT; (* Maximum number of dwords that can be processed *)
    tempDword : DINT; (* Temporary storage for building dword *)
    currentByteValue : DINT; (* Temporary storage for byte value *)
END_VAR
VAR CONSTANT
    BYTE_ARRAY_SIZE : DINT := 20; (* Size of the input byte array *)
    DWORD_ARRAY_SIZE : DINT := 10; (* Size of the output DINT array *)
END_VAR

(* Initialize output array and counter *)
FOR i := 1 TO DWORD_ARRAY_SIZE DO
    dwordArray[i] := 0;
END_FOR;
mergeDwordNum := 0;

(* Calculate maximum number of complete 4-byte chunks available *)
maxDwordCount := BYTE_ARRAY_SIZE / 4; (* Integer division truncates remainder *)

(* Limit processing by output array capacity *)
IF maxDwordCount > DWORD_ARRAY_SIZE THEN
    maxDwordCount := DWORD_ARRAY_SIZE;
END_IF;

(* Process each complete 4-byte chunk *)
dwordIdx := 1;
byteIdx := 1;
WHILE (dwordIdx <= maxDwordCount) DO
    tempDword := 0;

    (* Merge 4 bytes into one double word *)
    FOR j := 0 TO 3 DO
        currentByteValue := byteArray[byteIdx + j];

        (* Ensure byte value is in valid range (0-255) *)
        IF currentByteValue < 0 THEN
            currentByteValue := currentByteValue AND 16#000000FF;
        ELSIF currentByteValue > 255 THEN
            currentByteValue := currentByteValue AND 16#000000FF;
        END_IF;

        (* Shift byte into position and combine *)
        tempDword := tempDword OR SHL(currentByteValue, (j * 8));
    END_FOR;

    (* Store the merged double word *)
    dwordArray[dwordIdx] := tempDword;

    (* Update counters *)
    mergeDwordNum := mergeDwordNum + 1;
    dwordIdx := dwordIdx + 1;
    byteIdx := byteIdx + 4;
END_WHILE;

END_FUNCTION_BLOCK;

(* ---- hf_16.st ---- *)
TYPE
    ST_LinearSegment : STRUCT
        InputMin : REAL;
        InputMax : REAL;
        OutputMin : REAL;
        OutputMax : REAL;
    END_STRUCT;

    E_StatusCode : (
        STATUS_OK := 16#0000,
        STATUS_OUT_OF_RANGE := 16#8001
    );
END_TYPE

VAR_GLOBAL CONSTANT
    gc_Segments : ARRAY[1..3] OF ST_LinearSegment := [
        (InputMin := 1200.0, InputMax := 3600.0, OutputMin := 150.0, OutputMax := 240.0),
        (InputMin := 3600.0, InputMax := 4800.0, OutputMin := 240.0, OutputMax := 560.0),
        (InputMin := 4800.0, InputMax := 7000.0, OutputMin := 560.0, OutputMax := 720.0)
    ];
    gc_InputMinLimit : REAL := 1200.0;
    gc_InputMaxLimit : REAL := 7000.0;
    gc_OutputMinLimit : REAL := 150.0;
    gc_OutputMaxLimit : REAL := 720.0;
END_VAR

FUNCTION_BLOCK FB_LinearizeValue
VAR_INPUT
    InputValue : REAL;
END_VAR

VAR_OUTPUT
    LinearizedValue : REAL;
    Error : BOOL;
    Status : WORD;
END_VAR

VAR
    iSegmentIndex : INT;
    bValueProcessed : BOOL;
END_VAR

(* Initialize outputs *)
LinearizedValue := 0.0;
Error := FALSE;
Status := E_StatusCode.STATUS_OK;
bValueProcessed := FALSE;

(* Check for out-of-range conditions *)
IF InputValue < gc_InputMinLimit THEN
    LinearizedValue := gc_OutputMinLimit;
    Error := TRUE;
    Status := E_StatusCode.STATUS_OUT_OF_RANGE;
    bValueProcessed := TRUE;
ELSIF InputValue > gc_InputMaxLimit THEN
    LinearizedValue := gc_OutputMaxLimit;
    Error := TRUE;
    Status := E_StatusCode.STATUS_OUT_OF_RANGE;
    bValueProcessed := TRUE;
END_IF;

(* Process valid ranges if not already handled *)
IF NOT bValueProcessed THEN
    FOR iSegmentIndex := 1 TO 3 DO
        IF (InputValue >= gc_Segments[iSegmentIndex].InputMin)
           AND (InputValue <= gc_Segments[iSegmentIndex].InputMax) THEN
            LinearizedValue := gc_Segments[iSegmentIndex].OutputMin
                + (InputValue - gc_Segments[iSegmentIndex].InputMin)
                * (gc_Segments[iSegmentIndex].OutputMax - gc_Segments[iSegmentIndex].OutputMin)
                / (gc_Segments[iSegmentIndex].InputMax - gc_Segments[iSegmentIndex].InputMin);
            Error := FALSE;
            Status := E_StatusCode.STATUS_OK;
            bValueProcessed := TRUE;
            EXIT;
        END_IF;
    END_FOR;
END_IF;

(* Handle edge case: value within global limits but not in any segment *)
IF NOT bValueProcessed THEN
    LinearizedValue := 0.0;
    Error := TRUE;
    Status := E_StatusCode.STATUS_OUT_OF_RANGE;
END_IF;

END_FUNCTION_BLOCK;

(* ---- hf_17.st ---- *)
TYPE
    ST_WarehouseStatus :
        STRUCT
            productNum : INT;
            libFreeNum : INT;
            error : BOOL;
            status : WORD;
        END_STRUCT;
    ARRAY_StoragePositions : ARRAY[1..9] OF BOOL;
END_TYPE

FUNCTION_BLOCK FB_WarehouseManagement
VAR_INPUT
    requestIn : BOOL := FALSE;
    requestOut : BOOL := FALSE;
END_VAR

VAR_OUTPUT
    productNum : INT := 0;
    libFreeNum : INT := 9;
    error : BOOL := FALSE;
    status : WORD := 16#0000;
END_VAR

VAR_IN_OUT
    library : ARRAY_StoragePositions;
END_VAR

VAR
    i : INT;
    found : BOOL;
    errFull : WORD := 16#8001;
    errEmpty : WORD := 16#8002;
    initDone : BOOL := FALSE;
END_VAR

(* Reset error status at start of each cycle *)
error := FALSE;
status := 16#0000;

(* Initialize library array on first execution *)
IF NOT initDone THEN
    i := 1;
    WHILE i <= 9 DO
        library[i] := FALSE;
        i := i + 1;
    END_WHILE;
    initDone := TRUE;
END_IF;

(* Calculate current product count and free positions *)
productNum := 0;
i := 1;
WHILE i <= 9 DO
    IF library[i] THEN
        productNum := productNum + 1;
    END_IF;
    i := i + 1;
END_WHILE;
libFreeNum := 9 - productNum;

(* Handle product storage request *)
IF requestIn THEN
    (* Check for storage full condition *)
    IF productNum >= 9 THEN
        error := TRUE;
        status := errFull;
    ELSE
        (* Search for free position from highest to lowest index (FILO) *)
        found := FALSE;
        i := 9;
        WHILE i >= 1 AND NOT found DO
            IF NOT library[i] THEN
                library[i] := TRUE;
                found := TRUE;
            END_IF;
            i := i - 1;
        END_WHILE;

        (* Update counters if position was found *)
        IF found THEN
            productNum := productNum + 1;
            libFreeNum := libFreeNum - 1;
        END_IF;
    END_IF;
END_IF;

(* Handle product retrieval request *)
IF requestOut THEN
    (* Check for storage empty condition *)
    IF productNum <= 0 THEN
        error := TRUE;
        status := errEmpty;
    ELSE
        (* Search for occupied position from lowest to highest index (FIFO) *)
        found := FALSE;
        i := 1;
        WHILE i <= 9 AND NOT found DO
            IF library[i] THEN
                library[i] := FALSE;
                found := TRUE;
            END_IF;
            i := i + 1;
        END_WHILE;

        (* Update counters if position was found *)
        IF found THEN
            productNum := productNum - 1;
            libFreeNum := libFreeNum + 1;
        END_IF;
    END_IF;
END_IF;

(* Validate counter consistency - safety check *)
IF (productNum + libFreeNum) <> 9 THEN
    error := TRUE;
    status := 16#8003;  (* Internal consistency error *)
END_IF;

END_FUNCTION_BLOCK

(* ---- hf_18.st ---- *)
FUNCTION_BLOCK FB_ColorLightControl
{ S7_Optimized_Access := 'TRUE' }
VAR_INPUT
    controlButton : BOOL; // Push button for sequence control
END_VAR

VAR_OUTPUT
    greenLight : BOOL; // Green light control signal
    redLight : BOOL; // Red light control signal
    yellowLight : BOOL; // Yellow light control signal
END_VAR

VAR
    state : INT := 1; // State machine control variable
    lastControlButton : BOOL := FALSE; // Previous button state
END_VAR

// Main logic
IF controlButton AND NOT lastControlButton THEN
    // Rising edge detected - execute state transition
    CASE state OF
        1: // State 1: Green Only
            greenLight := TRUE;
            redLight := FALSE;
            yellowLight := FALSE;
            state := 2;

        2: // State 2: Red Only
            greenLight := FALSE;
            redLight := TRUE;
            yellowLight := FALSE;
            state := 3;

        3: // State 3: Yellow Only
            greenLight := FALSE;
            redLight := FALSE;
            yellowLight := TRUE;
            state := 4;

        4: // State 4: All Lights On
            greenLight := TRUE;
            redLight := TRUE;
            yellowLight := TRUE;
            state := 5;

        5: // State 5: All Lights Off
            greenLight := FALSE;
            redLight := FALSE;
            yellowLight := FALSE;
            state := 1;

        ELSE // Handle unexpected state (safety fallback)
            state := 1;
            greenLight := FALSE;
            redLight := FALSE;
            yellowLight := FALSE;
    END_CASE;
ELSE
    // No rising edge - maintain current state outputs
    CASE state OF
        1: // State 1: Green Only
            greenLight := TRUE;
            redLight := FALSE;
            yellowLight := FALSE;

        2: // State 2: Red Only
            greenLight := FALSE;
            redLight := TRUE;
            yellowLight := FALSE;

        3: // State 3: Yellow Only
            greenLight := FALSE;
            redLight := FALSE;
            yellowLight := TRUE;

        4: // State 4: All Lights On
            greenLight := TRUE;
            redLight := TRUE;
            yellowLight := TRUE;

        5: // State 5: All Lights Off
            greenLight := FALSE;
            redLight := FALSE;
            yellowLight := FALSE;

        ELSE // Safety fallback for unexpected state
            greenLight := FALSE;
            redLight := FALSE;
            yellowLight := FALSE;
    END_CASE;
END_IF;

// Update last button state for edge detection in next cycle
lastControlButton := controlButton;

END_FUNCTION_BLOCK;

(* ---- hf_19.st ---- *)
FUNCTION_BLOCK FB_DatabaseManager
VAR_INPUT
    dataInput : ARRAY[0..5] OF BYTE;
    storeTrigger : BOOL;
    resetTrigger : BOOL;
END_VAR

VAR_OUTPUT
    usedSpace : INT := 0;
    remainingSpace : INT := 20;
    error : BOOL;
    status : WORD;
END_VAR

VAR_IN_OUT
    dataBase : ARRAY[1..20] OF BYTE;
END_VAR

VAR
    dataLength : INT;
    i : INT;
END_VAR

(* Reset Operation - Highest Priority *)
IF resetTrigger THEN
    (* Clear database array *)
    FOR i := 1 TO 20 DO
        dataBase[i] := 0;
    END_FOR;

    (* Reset counters *)
    usedSpace := 0;
    remainingSpace := 20;

    (* Clear status *)
    error := FALSE;
    status := 0;

(* Store Operation - Conditional Execution *)
ELSIF storeTrigger THEN
    (* Extract and validate data length *)
    dataLength := dataInput[0];

    (* Length Validation *)
    IF (dataLength <= 0) OR (dataLength > 5) THEN
        error := TRUE;
        status := 16#8001;  (* Invalid data length *)

    (* Space Verification *)
    ELSIF (usedSpace + dataLength) > 20 THEN
        error := TRUE;
        status := 16#8002;  (* Insufficient space *)

    (* Data Storage *)
    ELSE
        (* Copy data bytes to database *)
        FOR i := 1 TO dataLength DO
            dataBase[usedSpace + i] := dataInput[i];
        END_FOR;

        (* Update space tracking *)
        usedSpace := usedSpace + dataLength;
        remainingSpace := 20 - usedSpace;

        (* Set success status *)
        error := FALSE;
        status := 0;
    END_IF;
END_IF;

END_FUNCTION_BLOCK

(* ---- hf_2.st ---- *)
(*
    FUNCTION_BLOCK: FindMinMaxValues
    Description: Finds the minimum and maximum values in a fixed-size array of integers
                and returns their values and positions (indices).
    Inputs:
        values : ARRAY[1..10] OF DINT - The array to be searched.
    Outputs:
        minValue : DINT - The minimum value found in the array.
        minValueIndex : DINT - The position (index) of the minimum value.
        maxValue : DINT - The maximum value found in the array.
        maxValueIndex : DINT - The position (index) of the maximum value.
    Implementation:
        Initializes min and max to the first element, then iterates through the
        remaining elements. Updates values and indices when a new min or max is found.
        Correctly handles edge cases (e.g., all elements equal, first element is min/max).
*)

FUNCTION_BLOCK FindMinMaxValues
VAR_INPUT
    values : ARRAY[1..10] OF DINT;
END_VAR
VAR_OUTPUT
    minValue : DINT;
    minValueIndex : DINT;
    maxValue : DINT;
    maxValueIndex : DINT;
END_VAR
VAR
    i : INT;
END_VAR

    (* Initialize with the first element *)
    minValue := values[1];
    maxValue := values[1];
    minValueIndex := 1;
    maxValueIndex := 1;

    (* Iterate through the rest of the array (elements 2 to 10) *)
    FOR i := 2 TO 10 DO
        IF values[i] < minValue THEN
            minValue := values[i];
            minValueIndex := i;
        END_IF;
        IF values[i] > maxValue THEN
            maxValue := values[i];
            maxValueIndex := i;
        END_IF;
    END_FOR;

END_FUNCTION_BLOCK;

(* ---- hf_20.st ---- *)
FUNCTION_BLOCK FB_ProductionLineControl
VAR_INPUT
    Mode : BOOL;            // Manual/Auto mode selection
    ForwardButton : BOOL;   // Forward rotation button
    ReverseButton : BOOL;   // Reverse rotation button
    SensorA : BOOL;         // Sensor A input
    SensorB : BOOL;         // Sensor B input
    SensorC : BOOL;         // Sensor C input
    ButtonA : BOOL;         // Button A input
    ButtonB : BOOL;         // Button B input
    ButtonC : BOOL;         // Button C input
END_VAR

VAR_OUTPUT
    MotorForward : BOOL;    // Motor forward output
    MotorReverse : BOOL;    // Motor reverse output
    CompletionLight : BOOL; // Process completion indicator
END_VAR

VAR
    State : INT := 0;       // State machine current state
END_VAR

// Main execution logic
CASE State OF
    0: // Initialization state
        MotorForward := FALSE;
        MotorReverse := FALSE;
        CompletionLight := FALSE;
        State := 1;

    1: // State 1: Waiting at Station A
        IF NOT Mode THEN // Manual Mode
            // Manual motor control with mutual exclusion
            IF ForwardButton AND NOT ReverseButton THEN
                MotorForward := TRUE;
                MotorReverse := FALSE;
            ELSIF ReverseButton AND NOT ForwardButton THEN
                MotorForward := FALSE;
                MotorReverse := TRUE;
            ELSE
                MotorForward := FALSE;
                MotorReverse := FALSE;
            END_IF;
            CompletionLight := FALSE;
        ELSE // Automatic Mode
            // Safety: Ensure reverse motor is off in auto mode
            MotorReverse := FALSE;
            MotorForward := FALSE;

            // Wait for SensorA activation
            IF SensorA THEN
                State := 2;
            END_IF;
        END_IF;

    2: // State 2: Processing at Station A
        IF NOT Mode THEN // Manual Mode
            IF ForwardButton AND NOT ReverseButton THEN
                MotorForward := TRUE;
                MotorReverse := FALSE;
            ELSIF ReverseButton AND NOT ForwardButton THEN
                MotorForward := FALSE;
                MotorReverse := TRUE;
            ELSE
                MotorForward := FALSE;
                MotorReverse := FALSE;
            END_IF;
            CompletionLight := FALSE;
        ELSE // Automatic Mode
            MotorReverse := FALSE;
            MotorForward := FALSE;

            // Wait for ButtonA press
            IF ButtonA THEN
                MotorForward := TRUE;
                State := 3;
            END_IF;
        END_IF;

    3: // State 3: Moving to Station B
        IF NOT Mode THEN // Manual Mode
            IF ForwardButton AND NOT ReverseButton THEN
                MotorForward := TRUE;
                MotorReverse := FALSE;
            ELSIF ReverseButton AND NOT ForwardButton THEN
                MotorForward := FALSE;
                MotorReverse := TRUE;
            ELSE
                MotorForward := FALSE;
                MotorReverse := FALSE;
            END_IF;
            CompletionLight := FALSE;
        ELSE // Automatic Mode
            MotorReverse := FALSE;

            // Wait for SensorB activation
            IF SensorB THEN
                MotorForward := FALSE;
                State := 4;
            END_IF;
        END_IF;

    4: // State 4: Processing at Station B
        IF NOT Mode THEN // Manual Mode
            IF ForwardButton AND NOT ReverseButton THEN
                MotorForward := TRUE;
                MotorReverse := FALSE;
            ELSIF ReverseButton AND NOT ForwardButton THEN
                MotorForward := FALSE;
                MotorReverse := TRUE;
            ELSE
                MotorForward := FALSE;
                MotorReverse := FALSE;
            END_IF;
            CompletionLight := FALSE;
        ELSE // Automatic Mode
            MotorReverse := FALSE;
            MotorForward := FALSE;

            // Wait for ButtonB press
            IF ButtonB THEN
                MotorForward := TRUE;
                State := 5;
            END_IF;
        END_IF;

    5: // State 5: Moving to Station C
        IF NOT Mode THEN // Manual Mode
            IF ForwardButton AND NOT ReverseButton THEN
                MotorForward := TRUE;
                MotorReverse := FALSE;
            ELSIF ReverseButton AND NOT ForwardButton THEN
                MotorForward := FALSE;
                MotorReverse := TRUE;
            ELSE
                MotorForward := FALSE;
                MotorReverse := FALSE;
            END_IF;
            CompletionLight := FALSE;
        ELSE // Automatic Mode
            MotorReverse := FALSE;

            // Wait for SensorC activation
            IF SensorC THEN
                MotorForward := FALSE;
                State := 6;
            END_IF;
        END_IF;

    6: // State 6: Processing at Station C
        IF NOT Mode THEN // Manual Mode
            IF ForwardButton AND NOT ReverseButton THEN
                MotorForward := TRUE;
                MotorReverse := FALSE;
            ELSIF ReverseButton AND NOT ForwardButton THEN
                MotorForward := FALSE;
                MotorReverse := TRUE;
            ELSE
                MotorForward := FALSE;
                MotorReverse := FALSE;
            END_IF;
            CompletionLight := FALSE;
        ELSE // Automatic Mode
            MotorReverse := FALSE;
            MotorForward := FALSE;

            // Wait for ButtonC press
            IF ButtonC THEN
                CompletionLight := TRUE;
                State := 7;
            END_IF;
        END_IF;

    7: // State 7: Cycle Completion
        IF NOT Mode THEN // Manual Mode
            IF ForwardButton AND NOT ReverseButton THEN
                MotorForward := TRUE;
                MotorReverse := FALSE;
            ELSIF ReverseButton AND NOT ForwardButton THEN
                MotorForward := FALSE;
                MotorReverse := TRUE;
            ELSE
                MotorForward := FALSE;
                MotorReverse := FALSE;
            END_IF;
            CompletionLight := FALSE;
        ELSE // Automatic Mode
            MotorReverse := FALSE;
            MotorForward := FALSE;

            // Wait for product removal (SensorC deactivation)
            IF NOT SensorC THEN
                CompletionLight := FALSE;
                State := 1;
            END_IF;
        END_IF;

END_CASE;

END_FUNCTION_BLOCK;

(* ---- hf_21.st ---- *)
FUNCTION_BLOCK FB_SplitNumber
VAR_INPUT
    InputNumber : INT;
END_VAR

VAR_OUTPUT
    Thousands : INT;
    Hundreds : INT;
    Tens : INT;
    Ones : INT;
    Min : INT;
    error : BOOL;
    status : WORD;
END_VAR

VAR
    tempNumber : INT;
    minValue : INT;
    digitProcessed : BOOL;
END_VAR

(* Input Validation *)
IF (InputNumber < 0) OR (InputNumber > 9999) THEN
    (* Error case: Input out of valid range *)
    error := TRUE;
    status := 16#8001;

    (* Zero all outputs *)
    Thousands := 0;
    Hundreds := 0;
    Tens := 0;
    Ones := 0;
    Min := 0;
ELSE
    (* Valid case: Normal operation *)
    error := FALSE;
    status := 16#0000;

    (* Digit Separation Logic *)
    tempNumber := InputNumber;
    Thousands := tempNumber / 1000;
    tempNumber := tempNumber MOD 1000;
    Hundreds := tempNumber / 100;
    tempNumber := tempNumber MOD 100;
    Tens := tempNumber / 10;
    Ones := tempNumber MOD 10;

    (* Minimum Non-Zero Digit Detection *)
    minValue := 0;
    digitProcessed := FALSE;

    (* Process each digit sequentially, excluding zeros *)
    IF Thousands <> 0 THEN
        minValue := Thousands;
        digitProcessed := TRUE;
    END_IF;

    IF Hundreds <> 0 THEN
        IF digitProcessed THEN
            minValue := minimal(minValue, Hundreds);
        ELSE
            minValue := Hundreds;
            digitProcessed := TRUE;
        END_IF;
    END_IF;

    IF Tens <> 0 THEN
        IF digitProcessed THEN
            minValue := minimal(minValue, Tens);
        ELSE
            minValue := Tens;
            digitProcessed := TRUE;
        END_IF;
    END_IF;

    IF Ones <> 0 THEN
        IF digitProcessed THEN
            minValue := minimal(minValue, Ones);
        ELSE
            minValue := Ones;
            digitProcessed := TRUE;
        END_IF;
    END_IF;

    (* Set final Min output *)
    IF NOT digitProcessed THEN
        (* All digits were zero *)
        Min := 0;
    ELSE
        Min := minValue;
    END_IF;
END_IF;

END_FUNCTION_BLOCK

(* Provided minimal function *)
FUNCTION minimal : INT
VAR_INPUT
    IN1 : INT;
    IN2 : INT;
END_VAR

IF IN1 <= IN2 THEN
    minimal := IN1;
ELSE
    minimal := IN2;
END_IF;

END_FUNCTION

(* ---- hf_3.st ---- *)
FUNCTION_BLOCK MultiPumpCtrl
VAR_INPUT
    mode : BOOL;                    (* FALSE = Manual, TRUE = Automatic *)
    start : BOOL;                   (* Start button *)
    stop : BOOL;                    (* Stop button - highest priority *)
    priorities : ARRAY[1..5] OF INT; (* Priority of each pump *)
    selections : ARRAY[1..5] OF BOOL; (* Manual selection for each pump *)
END_VAR

VAR_OUTPUT
    RunComds : ARRAY[1..5] OF BOOL; (* Run command for each pump *)
END_VAR

VAR
    i : INT;                        (* Loop counter *)
    j : INT;                        (* Loop counter *)
    maxPriority : INT;              (* Temporary variable for finding max priority *)
    maxIndex : INT;                 (* Index of pump with max priority *)
    runCount : INT;                 (* Counter for pumps selected in auto mode *)
    usedInAuto : ARRAY[1..5] OF BOOL; (* Tracks pumps already selected in auto mode *)
END_VAR

(* Main logic *)
IF stop THEN
    (* Stop has highest priority - stop all pumps *)
    FOR i := 1 TO 5 DO
        RunComds[i] := FALSE;
    END_FOR;
ELSE
    IF start THEN
        IF NOT mode THEN            (* Manual mode *)
            FOR i := 1 TO 5 DO
                RunComds[i] := selections[i];
            END_FOR;
        ELSE                        (* Automatic mode *)
            (* Initialize arrays *)
            FOR i := 1 TO 5 DO
                usedInAuto[i] := FALSE;
                RunComds[i] := FALSE;
            END_FOR;

            (* Find and run 3 pumps with highest priorities *)
            runCount := 0;
            WHILE runCount < 3 DO
                maxPriority := -32768;  (* Minimum INT value *)
                maxIndex := 0;

                (* Find the highest priority pump not already selected *)
                FOR i := 1 TO 5 DO
                    IF (priorities[i] > maxPriority) AND NOT usedInAuto[i] THEN
                        maxPriority := priorities[i];
                        maxIndex := i;
                    END_IF;
                END_FOR;

                (* If a pump was found (should always be true if runCount < 3) *)
                IF maxIndex > 0 THEN
                    RunComds[maxIndex] := TRUE;
                    usedInAuto[maxIndex] := TRUE;
                    runCount := runCount + 1;
                END_IF;
            END_WHILE;
        END_IF;
    ELSE                            (* start is FALSE *)
        FOR i := 1 TO 5 DO
            RunComds[i] := FALSE;
        END_FOR;
    END_IF;
END_IF;

END_FUNCTION_BLOCK;

(* ---- hf_4.st ---- *)
TYPE
    E_STATUS : (STATUS_OK := 0, STATUS_INVALID_YEAR := 16#8001, STATUS_INVALID_MONTH := 16#8002, STATUS_INVALID_DAY := 16#8003);
END_TYPE

FUNCTION_BLOCK FB_CalculateDayOfYear
VAR_INPUT
    Year : INT;
    Month : INT;
    Day : INT;
END_VAR

VAR_OUTPUT
    DayOfYear : INT;
    error : BOOL;
    status : WORD;
END_VAR

VAR
    DaysInMonth : ARRAY[1..12] OF INT := [31, 28, 31, 30, 31, 30, 31, 31, 30, 31, 30, 31];
END_VAR

VAR_TEMP
    i : INT;
    LeapYear : BOOL;
    MaxDay : INT;
END_VAR

    // Initialize outputs
    DayOfYear := 0;
    error := FALSE;
    status := WORD(STATUS_OK);

    // 1. Validate Month (highest priority)
    IF (Month < 1) OR (Month > 12) THEN
        error := TRUE;
        status := WORD(STATUS_INVALID_MONTH);
        RETURN;
    END_IF;

    // 2. Validate Day (second priority)
    // Check for positive value
    IF (Day <= 0) THEN
        error := TRUE;
        status := WORD(STATUS_INVALID_DAY);
        RETURN;
    END_IF;

    // Determine maximum days for the given month
    MaxDay := DaysInMonth[Month];
    IF (Month = 2) THEN
        // Calculate leap year for February validation
        LeapYear := ((Year MOD 4 = 0) AND (Year MOD 100 <> 0)) OR (Year MOD 400 = 0);
        IF LeapYear THEN
            MaxDay := 29;
        END_IF;
    END_IF;

    // Check if day exceeds maximum for the month
    IF (Day > MaxDay) THEN
        error := TRUE;
        status := WORD(STATUS_INVALID_DAY);
        RETURN;
    END_IF;

    // 3. Validate Year (lowest priority)
    IF (Year < 1000) OR (Year > 3000) THEN
        error := TRUE;
        status := WORD(STATUS_INVALID_YEAR);
        RETURN;
    END_IF;

    // All inputs are valid - proceed with calculation
    // Recalculate leap year for the final calculation
    LeapYear := ((Year MOD 4 = 0) AND (Year MOD 100 <> 0)) OR (Year MOD 400 = 0);

    // Start with the current day
    DayOfYear := Day;

    // Add days from all completed months
    FOR i := 1 TO (Month - 1) DO
        DayOfYear := DayOfYear + DaysInMonth[i];
    END_FOR;

    // Add extra day for leap year if date is after February
    IF (LeapYear AND (Month > 2)) THEN
        DayOfYear := DayOfYear + 1;
    END_IF;

END_FUNCTION_BLOCK

(* ---- hf_5.st ---- *)
TYPE
    SortStatus : WORD := 16#0000;
    SortErrorCode : WORD := 16#8A01;
END_TYPE

FUNCTION_BLOCK SelectSort
VAR_INPUT
    exe : BOOL;
    seq : ARRAY[1..100] OF INT;
END_VAR
VAR_OUTPUT
    error : BOOL;
    status : WORD;
END_VAR
VAR
    i : INT;
    j : INT;
    min_idx : INT;
    temp : INT;
    n : INT := 100;
    seq_local : ARRAY[1..100] OF INT;
    exe_prev : BOOL;
    sort_successful : BOOL;
END_VAR

(* Initialize outputs to error state *)
error := TRUE;
status := SortErrorCode;

(* Execute sorting on rising edge of exe *)
IF exe AND NOT exe_prev THEN
    (* Copy input array to local working array *)
    seq_local := seq;
    sort_successful := TRUE;

    (* Selection sort algorithm *)
    FOR i := 1 TO n-1 DO
        min_idx := i;
        FOR j := i+1 TO n DO
            IF seq_local[j] < seq_local[min_idx] THEN
                min_idx := j;
            END_IF;
        END_FOR;

        (* Swap elements if necessary *)
        IF min_idx <> i THEN
            temp := seq_local[i];
            seq_local[i] := seq_local[min_idx];
            seq_local[min_idx] := temp;
        END_IF;
    END_FOR;

    (* Verify sorting was successful *)
    sort_successful := TRUE;
    FOR i := 1 TO n-1 DO
        IF seq_local[i] > seq_local[i+1] THEN
            sort_successful := FALSE;
            EXIT;
        END_IF;
    END_FOR;

    (* Update outputs based on verification *)
    IF sort_successful THEN
        (* Copy sorted array back to output *)
        seq := seq_local;
        error := FALSE;
        status := SortStatus;
    ELSE
        (* Sorting verification failed *)
        error := TRUE;
        status := SortErrorCode;
    END_IF;
END_IF;

(* Store previous execution state *)
exe_prev := exe;

END_FUNCTION_BLOCK

(* ---- hf_6.st ---- *)
FUNCTION_BLOCK RandomNumberGenerator
VAR_INPUT
    minValue : DINT;
    maxValue : DINT;
    randomSeed_in : DINT;
END_VAR
VAR_OUTPUT
    error : BOOL;
    status : WORD;
    randomNumber : DINT;
END_VAR
VAR
    workingSeed : DINT;
    rangeSize : DINT;
    rawRandom : DINT;
    scaledRandom : DINT;
END_VAR
    (* Initialize outputs *)
    error := FALSE;
    status := 16#0000;
    randomNumber := 0;

    (* Validate input range *)
    IF minValue > maxValue THEN
        error := TRUE;
        status := 16#8200;
        randomNumber := 0;
        RETURN;
    END_IF;

    (* Prepare seed: ensure positive and non-zero *)
    workingSeed := randomSeed_in;
    IF workingSeed < 0 THEN
        workingSeed := workingSeed * (-1);
    END_IF;
    IF workingSeed = 0 THEN
        workingSeed := 1;
    END_IF;

    (* Generate random number within specified range *)
    rangeSize := maxValue - minValue + 1;
    rawRandom := MOD(workingSeed, 32749);
    scaledRandom := MOD(rawRandom, rangeSize);
    randomNumber := minValue + scaledRandom;

    (* Set success status *)
    error := FALSE;
    status := 16#0000;
END_FUNCTION_BLOCK

(* ---- hf_7.st ---- *)
(*
    FUNCTION_BLOCK AnalogBatchConverter
    Purpose: Batch conversion of analog input signals to engineering units.
    Processes up to 10 channels in parallel based on configuration arrays.

    Inputs:
        count (INT): Number of active channels to process (1..10).
        analogValues (ARRAY[1..10] OF REAL): Raw ADC input values per channel.

    Configuration/Output Arrays (Index 1..10):
        channel_enable (BOOL): Enable conversion for this channel.
        channel_hiLIM (REAL): Upper scaling limit for non-temperature mode.
        channel_loLIM (REAL): Lower scaling limit for non-temperature mode.
        channel_bipolar (BOOL): Input range flag (FALSE=Unipolar, TRUE=Bipolar).
        channel_measuringMode (INT): Conversion mode (0=Non-temp, 1=Std temp, 2=Climatic temp).
        channel_retVal (WORD): Status/error code per channel (0=OK).
        channel_outputValue (REAL): Converted output value in engineering units.

    Error Codes:
        16#8001: Invalid measuringMode value (not 0, 1, or 2).
        16#8002: Invalid scaling range (channel_hiLIM <= channel_loLIM).
*)

FUNCTION_BLOCK AnalogBatchConverter
VAR_INPUT
    count : INT;                            (* Number of channels to process (1..10) *)
    analogValues : ARRAY[1..10] OF REAL;    (* Raw ADC input values per channel *)
END_VAR

VAR_OUTPUT
    channel_enable : ARRAY[1..10] OF BOOL;      (* Enable flag per channel *)
    channel_hiLIM : ARRAY[1..10] OF REAL;       (* Upper scaling limit per channel *)
    channel_loLIM : ARRAY[1..10] OF REAL;       (* Lower scaling limit per channel *)
    channel_bipolar : ARRAY[1..10] OF BOOL;     (* Input range flag per channel *)
    channel_measuringMode : ARRAY[1..10] OF INT;(* Conversion mode per channel *)
    channel_retVal : ARRAY[1..10] OF WORD;      (* Status/error code per channel *)
    channel_outputValue : ARRAY[1..10] OF REAL; (* Converted output value per channel *)
END_VAR

VAR
    i : INT;                (* Loop counter *)
    rawValue : REAL;        (* Temporary storage for analog input *)
    hiLIM : REAL;           (* Temporary storage for high limit *)
    loLIM : REAL;           (* Temporary storage for low limit *)
    bipolar : BOOL;         (* Temporary storage for bipolar flag *)
    measuringMode : INT;    (* Temporary storage for measuring mode *)
    enable : BOOL;          (* Temporary storage for enable flag *)
    retVal : WORD;          (* Temporary storage for return value *)
    outputValue : REAL;     (* Temporary storage for output value *)
END_VAR

(* Main processing loop for all 10 channels *)
FOR i := 1 TO 10 DO
    (* Load configuration and input values for current channel *)
    enable := channel_enable[i];
    hiLIM := channel_hiLIM[i];
    loLIM := channel_loLIM[i];
    bipolar := channel_bipolar[i];
    measuringMode := channel_measuringMode[i];
    rawValue := analogValues[i];

    (* Initialize temporary variables for this channel *)
    retVal := 0;
    outputValue := 0.0;

    (* Process only if channel is within active count and enabled *)
    IF (i <= count) AND enable THEN
        CASE measuringMode OF
            0:  (* Non-temperature measurement - perform linear scaling *)
                IF hiLIM <= loLIM THEN
                    retVal := 16#8002;  (* Invalid scaling range error *)
                ELSE
                    IF bipolar THEN
                        (* Bipolar scaling: -27648.0 to 27648.0 maps to loLIM to hiLIM *)
                        outputValue := loLIM + ((rawValue + 27648.0) / (27648.0 * 2.0)) * (hiLIM - loLIM);
                    ELSE
                        (* Unipolar scaling: 0.0 to 27648.0 maps to loLIM to hiLIM *)
                        outputValue := loLIM + (rawValue / 27648.0) * (hiLIM - loLIM);
                    END_IF;
                END_IF;

            1:  (* Standard temperature measurement - divide by 10 *)
                outputValue := rawValue / 10.0;

            2:  (* Climatic temperature measurement - divide by 100 *)
                outputValue := rawValue / 100.0;

            ELSE
                (* Invalid measuring mode *)
                retVal := 16#8001;
        END_CASE;
    END_IF;

    (* Store results back to output arrays *)
    channel_retVal[i] := retVal;
    channel_outputValue[i] := outputValue;
END_FOR;

END_FUNCTION_BLOCK;

(* ---- hf_8.st ---- *)
FUNCTION_BLOCK FB_HexDigitAnalyzer
VAR_INPUT
    InputNumber : INT;
END_VAR
VAR_OUTPUT
    Thousands : INT;
    Hundreds : INT;
    Tens : INT;
    Ones : INT;
    MinDigit : INT;
    error : BOOL;
    status : WORD;
END_VAR
VAR
    tempMinValue : INT;
END_VAR

(* Input Validation *)
IF (InputNumber < 0) OR (InputNumber > 9999) THEN
    error := TRUE;
    status := 16#8001;
    Thousands := 0;
    Hundreds := 0;
    Tens := 0;
    Ones := 0;
    MinDigit := 0;
ELSE
    error := FALSE;
    status := 16#0000;

    (* Digit Separation Logic *)
    Thousands := InputNumber / 1000;
    Hundreds := (InputNumber MOD 1000) / 100;
    Tens := (InputNumber MOD 100) / 10;
    Ones := InputNumber MOD 10;

    (* Minimum Non-Zero Digit Detection *)
    tempMinValue := 32767; (* Maximum INT value *)

    IF Thousands <> 0 THEN
        tempMinValue := minimal(tempMinValue, Thousands);
    END_IF;

    IF Hundreds <> 0 THEN
        tempMinValue := minimal(tempMinValue, Hundreds);
    END_IF;

    IF Tens <> 0 THEN
        tempMinValue := minimal(tempMinValue, Tens);
    END_IF;

    IF Ones <> 0 THEN
        tempMinValue := minimal(tempMinValue, Ones);
    END_IF;

    (* Final MinDigit Assignment *)
    IF tempMinValue = 32767 THEN
        MinDigit := 0; (* All digits were zero *)
    ELSE
        MinDigit := tempMinValue;
    END_IF;
END_IF;

END_FUNCTION_BLOCK;

(* ---- hf_9.st ---- *)
TYPE
    // Direction enumeration for clarity
    SortDirectionEnum : (Ascending, Descending);
END_TYPE

FUNCTION_BLOCK ShellSortFB
VAR_INPUT
    // Input array to be sorted (fixed size 1000)
    arr : ARRAY[1..1000] OF DINT;
    // FALSE = Ascending, TRUE = Descending
    sortDirection : BOOL;
END_VAR
VAR_OUTPUT
    // Sorted output array
    sorted_arr : ARRAY[1..1000] OF DINT;
    // Error flag (TRUE = error occurred)
    error : BOOL;
    // Status code (16#0000 = OK)
    status : WORD;
END_VAR
VAR
    // Algorithm variables
    i : DINT;
    j : DINT;
    gap : DINT;
    temp : DINT;
    // Fixed array size constant
    n : DINT := 1000;
    // Internal direction flag (TRUE = sort ascending)
    sortAscending : BOOL;
END_VAR

// 1. Copy input array to output array
sorted_arr := arr;

// 2. Initialize outputs to default values
error := FALSE;
status := 16#0000;

// 3. Validate array size (fixed at 1000, but checks maintained for robustness)
IF n <= 1 THEN
    error := TRUE;
    status := 16#8200;  // Array size ≤ 1
    RETURN;
END_IF;

IF n > 1000 THEN
    error := TRUE;
    status := 16#8201;  // Array size > 1000
    RETURN;
END_IF;

// 4. Determine sort direction
// sortDirection = FALSE → Ascending → sortAscending = TRUE
// sortDirection = TRUE → Descending → sortAscending = FALSE
sortAscending := NOT sortDirection;

// 5. Shell Sort Algorithm
gap := n / 2;  // Initial gap size

WHILE gap > 0 DO
    i := gap + 1;  // Start from first element after gap

    WHILE i <= n DO
        temp := sorted_arr[i];
        j := i;

        // Inner loop: insertion sort for current gap
        WHILE (j > gap) AND (
            (sortAscending AND (sorted_arr[j - gap] > temp)) OR
            (NOT sortAscending AND (sorted_arr[j - gap] < temp))
        ) DO
            sorted_arr[j] := sorted_arr[j - gap];
            j := j - gap;
        END_WHILE;

        sorted_arr[j] := temp;
        i := i + 1;
    END_WHILE;

    gap := gap / 2;  // Reduce gap
END_WHILE;

// 6. Successful completion
error := FALSE;
status := 16#0000;

END_FUNCTION_BLOCK;

(* ---- med_22.st ---- *)
FUNCTION_BLOCK CottonCandyMachine
VAR_INPUT
    SugarLevel : REAL; (* Current sugar level measurement *)
    SpinningSpeed : INT; (* Desired spinning speed command *)
END_VAR
VAR_OUTPUT
    SugarFeeder : BOOL; (* Control signal for sugar feeding mechanism *)
    MotorSpeed : INT; (* Actual spinning motor speed output *)
END_VAR

(* Internal variables for threshold values *)
VAR
    rSugarThreshold : REAL := 10.0; (* Sugar level threshold for feeding *)
    iSpeedThreshold : INT := 0; (* Speed threshold for motor activation *)
END_VAR

(* Main control logic *)
(* Sugar feeder control: Activate when sugar level is below threshold *)
SugarFeeder := SugarLevel < rSugarThreshold;

(* Motor speed control: Set to input speed if positive, otherwise 0 *)
IF SpinningSpeed > iSpeedThreshold THEN
    MotorSpeed := SpinningSpeed;
ELSE
    MotorSpeed := 0;
END_IF;

END_FUNCTION_BLOCK

(* ---- med_23.st ---- *)
FUNCTION_BLOCK SmartIrrigationSystem
VAR_INPUT
    SoilMoistureSensor1 : REAL;
    SoilMoistureSensor2 : REAL;
    WeatherForecast : INT; (* 0: Sunny, 1: Rainy, 2: Cloudy *)
END_VAR

VAR_OUTPUT
    WaterPump : BOOL;
END_VAR

VAR
    SoilMoistureThreshold : REAL := 30.0;
    bRainCondition : BOOL;
    bSunnyCondition : BOOL;
    bSoilDryCondition : BOOL;
    bPumpActivateCondition : BOOL;
END_VAR

(* Priority 1: Immediate deactivation for rainy forecast *)
bRainCondition := (WeatherForecast = 1);
IF bRainCondition THEN
    WaterPump := FALSE;
    RETURN;
END_IF;

(* Priority 2: Check activation conditions for sunny weather *)
bSunnyCondition := (WeatherForecast = 0);
bSoilDryCondition := (SoilMoistureSensor1 < SoilMoistureThreshold) OR (SoilMoistureSensor2 < SoilMoistureThreshold);
bPumpActivateCondition := bSunnyCondition AND bSoilDryCondition;

(* Set pump state based on activation conditions *)
IF bPumpActivateCondition THEN
    WaterPump := TRUE;
ELSE
    WaterPump := FALSE;
END_IF;

END_FUNCTION_BLOCK

(* ---- med_24.st ---- *)
(* ===================================================================== *)
(* FUNCTION_BLOCK: AutomaticDoorControl                                  *)
(* Description: Controls an automatic door for a retail environment.     *)
(*              The door opens on a rising edge of the proximity sensor  *)
(*              and remains open while the sensor is active or until a   *)
(*              fixed timer expires after the sensor becomes inactive.   *)
(* ===================================================================== *)
FUNCTION_BLOCK AutomaticDoorControl
VAR_INPUT
    ProximitySensor : BOOL; (* TRUE when an object is detected near the door *)
    ElapsedTime : DINT;     (* Time in milliseconds since the door was last opened *)
END_VAR

VAR_OUTPUT
    DoorOpen : BOOL;        (* TRUE to command the door open, FALSE to close *)
END_VAR

VAR
    (* Configuration Constant *)
    DoorOpenDuration : DINT := 5000; (* Time door stays open after sensor goes inactive [ms] *)

    (* Internal State Variables *)
    eCurrentState : (STATE_CLOSED, STATE_OPENING, STATE_OPEN, STATE_CLOSING) := STATE_CLOSED;
    tonOpenTimer : TON; (* Timer to manage the hold-open duration *)
    rTrigSensor : R_TRIG; (* Edge detector for the proximity sensor *)
END_VAR

(* --------------------------------------------------------------------- *)
(* Main State Machine Logic                                              *)
(* --------------------------------------------------------------------- *)
(* Detect rising edge of the sensor for clean activation *)
rTrigSensor(CLK := ProximitySensor);

CASE eCurrentState OF
    STATE_CLOSED:
        DoorOpen := FALSE;
        tonOpenTimer(IN := FALSE, PT := DINT_TO_TIME(DoorOpenDuration));

        (* Transition to OPENING on a rising edge of the sensor *)
        IF rTrigSensor.Q THEN
            eCurrentState := STATE_OPENING;
        END_IF;

    STATE_OPENING:
        (* Command the door to open and start the hold-open timer *)
        DoorOpen := TRUE;
        tonOpenTimer(IN := TRUE, PT := DINT_TO_TIME(DoorOpenDuration));
        eCurrentState := STATE_OPEN;

    STATE_OPEN:
        DoorOpen := TRUE;

        (* Check exit conditions from the OPEN state *)
        IF NOT ProximitySensor AND tonOpenTimer.Q THEN
            (* Sensor is inactive AND the hold timer has expired *)
            eCurrentState := STATE_CLOSING;
        ELSIF ProximitySensor THEN
            (* Sensor is still active: reset and restart the hold timer *)
            tonOpenTimer(IN := FALSE);
            tonOpenTimer(IN := TRUE, PT := DINT_TO_TIME(DoorOpenDuration));
        END_IF;
        (* If sensor is inactive but timer is still running, remain in STATE_OPEN *)

    STATE_CLOSING:
        (* Command the door to close and reset internal logic *)
        DoorOpen := FALSE;
        tonOpenTimer(IN := FALSE);
        eCurrentState := STATE_CLOSED;

END_CASE;

END_FUNCTION_BLOCK

(* ---- med_25.st ---- *)
FUNCTION_BLOCK WastewaterControl
VAR_INPUT
    InFlow : REAL;
    OutFlow : REAL;
    pH : REAL;
    TankLvl : REAL;
END_VAR

VAR_OUTPUT
    Pump1 : BOOL;
    Pump2 : BOOL;
    Valve1 : BOOL;
    Valve2 : BOOL;
END_VAR

VAR
    LowInFlow : REAL := 100.0;
    HighOutFlow : REAL := 90.0;
    DesiredPH : REAL := 7.0;
    HighTankLvl : REAL := 80.0;
END_VAR

// Control logic executed at each PLC cycle
Pump1 := InFlow < LowInFlow;
Pump2 := OutFlow > HighOutFlow;
Valve1 := pH < DesiredPH;
Valve2 := TankLvl > HighTankLvl;

END_FUNCTION_BLOCK

(* ---- med_26.st ---- *)
FUNCTION_BLOCK BookSorting
VAR_INPUT
    RFID1 : BOOL;
    RFID2 : BOOL;
    RFID3 : BOOL;
END_VAR

VAR_OUTPUT
    Motor : BOOL;
    Bin1 : BOOL;
    Bin2 : BOOL;
    Bin3 : BOOL;
END_VAR

// Main logic
Motor := RFID1 OR RFID2 OR RFID3;

IF RFID1 THEN
    Bin1 := TRUE;
    Bin2 := FALSE;
    Bin3 := FALSE;
ELSIF RFID2 THEN
    Bin1 := FALSE;
    Bin2 := TRUE;
    Bin3 := FALSE;
ELSIF RFID3 THEN
    Bin1 := FALSE;
    Bin2 := FALSE;
    Bin3 := TRUE;
ELSE
    Bin1 := FALSE;
    Bin2 := FALSE;
    Bin3 := FALSE;
END_IF;

END_FUNCTION_BLOCK

(* ---- med_27.st ---- *)
FUNCTION_BLOCK FlowerArrangingMachine
VAR_INPUT
    FlowerTypeSensor : INT; (* Input for detecting flower type *)
    FlowerColorSensor : INT; (* Input for detecting flower color *)
END_VAR
VAR_OUTPUT
    ArrangingMechanism : INT; (* Output for controlling arranging mechanism *)
    ConveyorBelt : BOOL; (* Output for controlling conveyor belt *)
END_VAR
VAR
    (* No internal variables required for this deterministic logic *)
END_VAR

(* Main control logic executed each PLC cycle *)
IF (FlowerTypeSensor = 1) AND (FlowerColorSensor = 1) THEN
    ArrangingMechanism := 1; (* Red type 1 flower *)
ELSIF (FlowerTypeSensor = 1) AND (FlowerColorSensor = 2) THEN
    ArrangingMechanism := 2; (* Blue type 1 flower *)
ELSIF (FlowerTypeSensor = 2) AND (FlowerColorSensor = 1) THEN
    ArrangingMechanism := 3; (* Red type 2 flower *)
ELSIF (FlowerTypeSensor = 2) AND (FlowerColorSensor = 2) THEN
    ArrangingMechanism := 4; (* Blue type 2 flower *)
ELSE
    ArrangingMechanism := 0; (* Any other combination *)
END_IF;

(* Conveyor belt control derived from arranging mechanism state *)
ConveyorBelt := (ArrangingMechanism <> 0);

END_FUNCTION_BLOCK;

(* ---- med_28.st ---- *)
FUNCTION_BLOCK HomeBrewingSystem
VAR_INPUT
    TemperatureSensor : REAL;     (* Current temperature measurement in °C *)
    WaterFlowSensor : REAL;       (* Current water flow measurement in units *)
    BrewingStartTime : TIME;      (* Absolute start time of brewing process *)
    BrewingDuration : TIME;       (* Total duration of brewing process *)
END_VAR
VAR_OUTPUT
    HeatingElement : BOOL;        (* Control signal for heating element *)
    AgitationMotor : BOOL;        (* Control signal for agitation motor *)
    HopsDispenser : BOOL;         (* Control signal for hops dispenser *)
    FermentationTank : BOOL;      (* Control signal for fermentation tank *)
END_VAR
VAR
    CurrentTime : TIME;           (* Current system time *)
    ElapsedBrewingTime : TIME;    (* Time elapsed since brewing started *)
    IsBrewingActive : BOOL;       (* Flag indicating if brewing is in progress *)
END_VAR

(* Calculate current time and elapsed brewing time *)
CurrentTime := TIME();
ElapsedBrewingTime := CurrentTime - BrewingStartTime;

(* Determine if brewing process is active *)
IsBrewingActive := (ElapsedBrewingTime >= T#0s) AND (ElapsedBrewingTime <= BrewingDuration);

(* Control heating element based on temperature *)
IF IsBrewingActive THEN
    HeatingElement := TemperatureSensor < 65.0;
ELSE
    HeatingElement := FALSE;
END_IF;

(* Control agitation motor based on water flow *)
IF IsBrewingActive THEN
    AgitationMotor := WaterFlowSensor > 0.5;
ELSE
    AgitationMotor := FALSE;
END_IF;

(* Control hops dispenser - activate after 5 hours *)
IF IsBrewingActive THEN
    HopsDispenser := ElapsedBrewingTime >= T#5h;
ELSE
    HopsDispenser := FALSE;
END_IF;

(* Control fermentation tank - activate after 48 hours *)
IF IsBrewingActive THEN
    FermentationTank := ElapsedBrewingTime >= T#48h;
ELSE
    FermentationTank := FALSE;
END_IF;

END_FUNCTION_BLOCK

(* ---- med_29.st ---- *)
(*
    FUNCTION_BLOCK: DocumentFilingSystem
    DESCRIPTION: Controls an automatic document filing system.
    LOGIC:
        - Conveyor motor runs when a document is detected AND a valid category (1-4) is selected.
        - Only the storage bin corresponding to the selected category is activated.
        - All outputs are deactivated when no document is detected OR an invalid category is selected.
    INPUTS:
        DocumentInlet : BOOL - Signal indicating a document is present at the inlet.
        CategorySelector : INT - Integer code (1-4) selecting the target storage bin.
    OUTPUTS:
        ConveyorMotor : BOOL - Control signal for the conveyor motor.
        StorageBin1 : BOOL - Control signal for storage bin 1 (Category 1).
        StorageBin2 : BOOL - Control signal for storage bin 2 (Category 2).
        StorageBin3 : BOOL - Control signal for storage bin 3 (Category 3).
        StorageBin4 : BOOL - Control signal for storage bin 4 (Category 4).
*)

FUNCTION_BLOCK DocumentFilingSystem
VAR_INPUT
    DocumentInlet : BOOL; (* Input to detect the arrival of a document *)
    CategorySelector : INT; (* Input to select the document category *)
END_VAR
VAR_OUTPUT
    ConveyorMotor : BOOL; (* Output to control the conveyor motor *)
    StorageBin1 : BOOL; (* Output to activate storage bin 1 *)
    StorageBin2 : BOOL; (* Output to activate storage bin 2 *)
    StorageBin3 : BOOL; (* Output to activate storage bin 3 *)
    StorageBin4 : BOOL; (* Output to activate storage bin 4 *)
END_VAR
VAR
    bValidCategory : BOOL; (* Internal flag for category validation *)
END_VAR

    (* 1. Validate the category selector input *)
    bValidCategory := (CategorySelector >= 1) AND (CategorySelector <= 4);

    (* 2. Main Control Logic: Activate outputs only if document is present AND category is valid *)
    IF DocumentInlet AND bValidCategory THEN
        (* Activate the conveyor motor *)
        ConveyorMotor := TRUE;

        (* Activate exactly one storage bin based on the CategorySelector *)
        CASE CategorySelector OF
            1:
                StorageBin1 := TRUE;
                StorageBin2 := FALSE;
                StorageBin3 := FALSE;
                StorageBin4 := FALSE;
            2:
                StorageBin1 := FALSE;
                StorageBin2 := TRUE;
                StorageBin3 := FALSE;
                StorageBin4 := FALSE;
            3:
                StorageBin1 := FALSE;
                StorageBin2 := FALSE;
                StorageBin3 := TRUE;
                StorageBin4 := FALSE;
            4:
                StorageBin1 := FALSE;
                StorageBin2 := FALSE;
                StorageBin3 := FALSE;
                StorageBin4 := TRUE;
            ELSE
                (* This branch is logically unreachable due to the bValidCategory check,
                   but included for robustness and completeness. *)
                StorageBin1 := FALSE;
                StorageBin2 := FALSE;
                StorageBin3 := FALSE;
                StorageBin4 := FALSE;
        END_CASE;
    ELSE
        (* 3. Deactivate all outputs if no document OR invalid category *)
        ConveyorMotor := FALSE;
        StorageBin1 := FALSE;
        StorageBin2 := FALSE;
        StorageBin3 := FALSE;
        StorageBin4 := FALSE;
    END_IF;

END_FUNCTION_BLOCK

(* ---- med_30.st ---- *)
FUNCTION_BLOCK MuseumClimateControl
VAR_INPUT
    HumiditySensor : REAL;
    TemperatureSensor : REAL;
    LightSensor : BOOL;
END_VAR

VAR_OUTPUT
    HVACSystem : BOOL;
    Humidifier : BOOL;
    Dehumidifier : BOOL;
    LightControl : BOOL;
END_VAR

VAR
    TargetHumidity : REAL := 50.0;
    TargetTemperature : REAL := 20.0;
    LightThreshold : BOOL := TRUE;
END_VAR

(* Humidity Control Logic *)
IF HumiditySensor < TargetHumidity THEN
    Humidifier := TRUE;
    Dehumidifier := FALSE;
ELSIF HumiditySensor > TargetHumidity THEN
    Humidifier := FALSE;
    Dehumidifier := TRUE;
ELSE
    Humidifier := FALSE;
    Dehumidifier := FALSE;
END_IF;

(* Temperature Control Logic *)
IF TemperatureSensor <> TargetTemperature THEN
    HVACSystem := TRUE;
ELSE
    HVACSystem := FALSE;
END_IF;

(* Lighting Control Logic *)
IF LightSensor AND LightThreshold THEN
    LightControl := FALSE;
ELSE
    LightControl := TRUE;
END_IF;

END_FUNCTION_BLOCK

(* ---- med_31.st ---- *)
FUNCTION_BLOCK ChargingStationControl
VAR_INPUT
    EVConnected : BOOL;
    EVVoltage : REAL;
    EVCurrent : REAL;
    EVStateOfCharge : REAL;
    ChargingTimer : TIME;
END_VAR

VAR_OUTPUT
    EVCharging : BOOL;
END_VAR

VAR
    VoltageOK : BOOL;
    CurrentOK : BOOL;
    SOCNotFull : BOOL;
    TimerOK : BOOL;
END_VAR

(* Evaluate all conditions using intermediate variables *)
VoltageOK := EVVoltage > 350.0;
CurrentOK := EVCurrent <= 32.0;
SOCNotFull := EVStateOfCharge < 100.0;
TimerOK := ChargingTimer <= T#2h;

(* Control logic: Start charging only when ALL conditions are met *)
IF EVConnected AND VoltageOK AND CurrentOK AND SOCNotFull AND TimerOK THEN
    EVCharging := TRUE;
ELSE
    EVCharging := FALSE;
END_IF;

END_FUNCTION_BLOCK

(* ---- med_32.st ---- *)
(* Greenhouse Watering System FUNCTION_BLOCK *)
(* Implements hysteresis control with 30% activation and 70% deactivation thresholds *)
(* Includes configurable response delay for state transitions *)

FUNCTION_BLOCK GreenhouseWateringSystem
VAR_INPUT
    SoilMoistureSensor : REAL; (* Input: Current soil moisture reading (0-100%) *)
    EnableSystem : BOOL := TRUE; (* Input: Master enable for the system *)
    ResponseDelay : TIME := T#5s; (* Input: Configurable delay for state transitions *)
END_VAR

VAR_OUTPUT
    SprinklersOn : BOOL := FALSE; (* Output: Control signal for sprinkler activation *)
    SystemState : INT := 0; (* Output: Current state of the system (0=Idle, 1=Activating, 2=Active, 3=Deactivating) *)
    LastMoistureReading : REAL := 0.0; (* Output: Last valid moisture reading *)
END_VAR

VAR
    (* Internal state variables *)
    CurrentState : INT := 0; (* 0=IDLE, 1=ACTIVATING, 2=ACTIVE, 3=DEACTIVATING *)

    (* Timer for response delay *)
    TransitionTimer : TON;

    (* Configuration constants *)
    LOW_THRESHOLD : REAL := 30.0; (* Activation threshold *)
    HIGH_THRESHOLD : REAL := 70.0; (* Deactivation threshold *)

    (* Internal flags *)
    TimerActive : BOOL := FALSE;
END_VAR

(* Main state machine logic *)
IF NOT EnableSystem THEN
    (* System disabled - reset to safe state *)
    SprinklersOn := FALSE;
    CurrentState := 0;
    TransitionTimer(IN:=FALSE, PT:=ResponseDelay);
    SystemState := CurrentState;
    RETURN;
END_IF;

(* Update last moisture reading for monitoring *)
LastMoistureReading := SoilMoistureSensor;

(* State machine implementation *)
CASE CurrentState OF
    0: (* IDLE STATE - Sprinklers are OFF *)
        SprinklersOn := FALSE;
        TransitionTimer(IN:=FALSE, PT:=ResponseDelay);
        TimerActive := FALSE;

        (* Check if moisture has dropped below activation threshold *)
        IF SoilMoistureSensor < LOW_THRESHOLD THEN
            CurrentState := 1; (* Transition to ACTIVATING state *)
            TransitionTimer(IN:=TRUE, PT:=ResponseDelay);
            TimerActive := TRUE;
        END_IF;

    1: (* ACTIVATING STATE - Waiting for delay before turning sprinklers ON *)
        SprinklersOn := FALSE;

        (* Continue timing if timer is active *)
        IF TimerActive THEN
            TransitionTimer(IN:=TRUE, PT:=ResponseDelay);

            (* Check if timer has completed *)
            IF TransitionTimer.Q THEN
                CurrentState := 2; (* Transition to ACTIVE state *)
                SprinklersOn := TRUE;
                TransitionTimer(IN:=FALSE, PT:=ResponseDelay);
                TimerActive := FALSE;
            END_IF;
        ELSE
            (* Timer was not properly started - restart it *)
            TransitionTimer(IN:=TRUE, PT:=ResponseDelay);
            TimerActive := TRUE;
        END_IF;

        (* Safety check: If moisture rises above activation threshold during delay, cancel activation *)
        IF SoilMoistureSensor >= LOW_THRESHOLD THEN
            CurrentState := 0; (* Return to IDLE state *)
            TransitionTimer(IN:=FALSE, PT:=ResponseDelay);
            TimerActive := FALSE;
            SprinklersOn := FALSE;
        END_IF;

    2: (* ACTIVE STATE - Sprinklers are ON *)
        SprinklersOn := TRUE;
        TransitionTimer(IN:=FALSE, PT:=ResponseDelay);
        TimerActive := FALSE;

        (* Check if moisture has risen above deactivation threshold *)
        IF SoilMoistureSensor > HIGH_THRESHOLD THEN
            CurrentState := 3; (* Transition to DEACTIVATING state *)
            TransitionTimer(IN:=TRUE, PT:=ResponseDelay);
            TimerActive := TRUE;
        END_IF;

    3: (* DEACTIVATING STATE - Waiting for delay before turning sprinklers OFF *)
        SprinklersOn := TRUE;

        (* Continue timing if timer is active *)
        IF TimerActive THEN
            TransitionTimer(IN:=TRUE, PT:=ResponseDelay);

            (* Check if timer has completed *)
            IF TransitionTimer.Q THEN
                CurrentState := 0; (* Transition to IDLE state *)
                SprinklersOn := FALSE;
                TransitionTimer(IN:=FALSE, PT:=ResponseDelay);
                TimerActive := FALSE;
            END_IF;
        ELSE
            (* Timer was not properly started - restart it *)
            TransitionTimer(IN:=TRUE, PT:=ResponseDelay);
            TimerActive := TRUE;
        END_IF;

        (* Safety check: If moisture drops below deactivation threshold during delay, cancel deactivation *)
        IF SoilMoistureSensor <= HIGH_THRESHOLD THEN
            CurrentState := 2; (* Return to ACTIVE state *)
            TransitionTimer(IN:=FALSE, PT:=ResponseDelay);
            TimerActive := FALSE;
            SprinklersOn := TRUE;
        END_IF;

    ELSE
        (* Error state - reset to safe IDLE state *)
        CurrentState := 0;
        SprinklersOn := FALSE;
        TransitionTimer(IN:=FALSE, PT:=ResponseDelay);
        TimerActive := FALSE;

END_CASE;

(* Update output state for monitoring *)
SystemState := CurrentState;

(* Assertion checks for system safety *)
(* Emergency shutoff if moisture exceeds maximum safe limit *)
IF SoilMoistureSensor > 95.0 THEN
    SprinklersOn := FALSE;
    CurrentState := 0;
    TransitionTimer(IN:=FALSE, PT:=ResponseDelay);
    TimerActive := FALSE;
END_IF;

(* Emergency activation if moisture drops below critical minimum *)
IF SoilMoistureSensor < 5.0 THEN
    SprinklersOn := TRUE;
    CurrentState := 2;
    TransitionTimer(IN:=FALSE, PT:=ResponseDelay);
    TimerActive := FALSE;
END_IF;

END_FUNCTION_BLOCK;

(* ---- med_33.st ---- *)
FUNCTION_BLOCK RoboticArmColorSorting
VAR_INPUT
    ColorSensorRed : BOOL;   (* Input: Red color sensor *)
    ColorSensorGreen : BOOL;  (* Input: Green color sensor *)
    ColorSensorBlue : BOOL;   (* Input: Blue color sensor *)
END_VAR

VAR_OUTPUT
    RoboticArmMove : BOOL := FALSE;     (* Output: Control for robotic arm movement *)
    BinRed : BOOL := FALSE;           (* Output: Activate red bin *)
    BinGreen : BOOL := FALSE;         (* Output: Activate green bin *)
    BinBlue : BOOL := FALSE;          (* Output: Activate blue bin *)
END_VAR

VAR
    bAnyColorDetected : BOOL;
END_VAR

(* Determine if any color is detected *)
bAnyColorDetected := ColorSensorRed OR ColorSensorGreen OR ColorSensorBlue;

(* Control robotic arm movement: activate when any color is detected *)
RoboticArmMove := bAnyColorDetected;

(* Control bin activation based on color detection *)
(* Only one bin is active at a time, with priority if multiple sensors are active *)
(* Priority order: Red, Green, Blue *)
IF ColorSensorRed THEN
    BinRed := TRUE;
    BinGreen := FALSE;
    BinBlue := FALSE;
ELSIF ColorSensorGreen THEN
    BinRed := FALSE;
    BinGreen := TRUE;
    BinBlue := FALSE;
ELSIF ColorSensorBlue THEN
    BinRed := FALSE;
    BinGreen := FALSE;
    BinBlue := TRUE;
ELSE
    BinRed := FALSE;
    BinGreen := FALSE;
    BinBlue := FALSE;
END_IF;

END_FUNCTION_BLOCK
